Yaskawa INFORM job: DEMO_ROOF_SIDE_0625_3PAINT_32.JBI

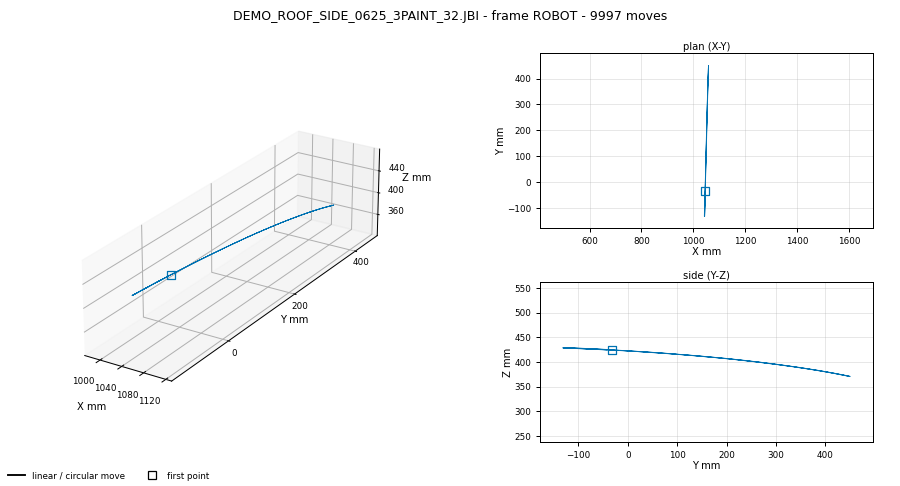
[picture p0: tool path of DEMO_ROOF_SIDE_0625_3PAINT_32.JBI in frame ROBOT, 9997 of 9997 moves have a stored position in this frame; points joined in program order, loops and branches not executed]
/JOB
//NAME DEMO_ROOF_SIDE_0625_3PAINT32
//POS
///NPOS 9997,0,0,0,0,0
///TOOL 0
///USER 0
///POSTYPE ROBOT
///RECTAN
///RCONF 1,0,0,0,0,0,0,0,0,0,0,0,0,0,0,0,0,0,0,0,0,0,0,0
C00000=1046.643,-32.584,425.197,169.918,33.552,156.330
C00001=1046.637,-32.833,425.210,169.916,33.551,156.330
C00002=1046.631,-33.082,425.224,169.914,33.549,156.330
C00003=1046.625,-33.331,425.237,169.912,33.548,156.330
C00004=1046.618,-33.581,425.250,169.910,33.547,156.329
C00005=1046.612,-33.831,425.264,169.908,33.546,156.329
C00006=1046.606,-34.081,425.276,169.906,33.544,156.329
C00007=1046.600,-34.330,425.290,169.904,33.543,156.329
C00008=1046.593,-34.580,425.303,169.902,33.542,156.329
C00009=1046.586,-34.860,425.319,169.899,33.541,156.329
C00010=1046.579,-35.141,425.334,169.897,33.539,156.329
C00011=1046.572,-35.422,425.348,169.895,33.538,156.328
C00012=1046.566,-35.702,425.363,169.893,33.536,156.328
C00013=1046.559,-35.952,425.377,169.891,33.535,156.328
C00014=1046.553,-36.202,425.389,169.889,33.534,156.328
C00015=1046.547,-36.451,425.403,169.887,33.533,156.328
C00016=1046.541,-36.700,425.416,169.885,33.531,156.328
C00017=1046.534,-36.950,425.429,169.883,33.530,156.327
C00018=1046.528,-37.200,425.442,169.881,33.529,156.327
C00019=1046.522,-37.450,425.455,169.879,33.528,156.327
C00020=1046.515,-37.699,425.469,169.877,33.526,156.327
C00021=1046.510,-37.949,425.481,169.875,33.525,156.327
C00022=1046.503,-38.198,425.494,169.873,33.524,156.327
C00023=1046.497,-38.447,425.508,169.870,33.523,156.326
C00024=1046.491,-38.698,425.521,169.868,33.521,156.326
C00025=1046.484,-38.947,425.534,169.866,33.520,156.326
C00026=1046.478,-39.196,425.547,169.864,33.519,156.326
C00027=1046.472,-39.446,425.560,169.862,33.518,156.326
C00028=1046.466,-39.695,425.573,169.860,33.517,156.326
C00029=1046.458,-39.945,425.586,169.858,33.515,156.326
C00030=1046.453,-40.195,425.599,169.856,33.515,156.325
C00031=1046.446,-40.444,425.612,169.854,33.513,156.325
C00032=1046.440,-40.694,425.624,169.852,33.512,156.325
C00033=1046.434,-40.943,425.638,169.850,33.511,156.325
C00034=1046.428,-41.193,425.650,169.848,33.510,156.325
C00035=1046.421,-41.443,425.663,169.846,33.509,156.325
C00036=1046.415,-41.692,425.677,169.844,33.507,156.325
C00037=1046.409,-41.942,425.689,169.842,33.507,156.324
C00038=1046.402,-42.191,425.702,169.840,33.505,156.324
C00039=1046.397,-42.441,425.715,169.838,33.504,156.324
C00040=1046.390,-42.690,425.728,169.836,33.503,156.324
C00041=1046.384,-42.940,425.740,169.834,33.502,156.324
C00042=1046.377,-43.189,425.753,169.832,33.501,156.324
C00043=1046.371,-43.440,425.766,169.830,33.500,156.324
C00044=1046.365,-43.689,425.780,169.827,33.498,156.324
C00045=1046.358,-43.939,425.792,169.825,33.497,156.323
C00046=1046.352,-44.188,425.805,169.823,33.496,156.323
C00047=1046.346,-44.438,425.817,169.821,33.495,156.323
C00048=1046.340,-44.687,425.831,169.819,33.494,156.323
C00049=1046.334,-44.937,425.843,169.817,33.493,156.323
C00050=1046.327,-45.187,425.855,169.815,33.492,156.323
C00051=1046.321,-45.436,425.868,169.813,33.490,156.323
C00052=1046.315,-45.686,425.881,169.811,33.490,156.322
C00053=1046.309,-45.935,425.894,169.809,33.488,156.322
C00054=1046.302,-46.185,425.906,169.807,33.487,156.322
C00055=1046.296,-46.435,425.919,169.805,33.486,156.322
C00056=1046.290,-46.684,425.932,169.803,33.485,156.322
C00057=1046.284,-46.934,425.945,169.801,33.484,156.322
C00058=1046.277,-47.183,425.958,169.799,33.483,156.322
C00059=1046.271,-47.433,425.970,169.797,33.482,156.321
C00060=1046.265,-47.683,425.983,169.794,33.481,156.321
C00061=1046.259,-47.932,425.996,169.792,33.479,156.321
C00062=1046.252,-48.182,426.008,169.790,33.478,156.321
C00063=1046.246,-48.432,426.021,169.788,33.477,156.321
C00064=1046.240,-48.681,426.034,169.786,33.476,156.321
C00065=1046.234,-48.931,426.046,169.784,33.475,156.321
C00066=1046.227,-49.181,426.058,169.782,33.474,156.321
C00067=1046.221,-49.430,426.072,169.780,33.473,156.320
C00068=1046.215,-49.680,426.084,169.778,33.472,156.320
C00069=1046.209,-49.930,426.097,169.776,33.470,156.320
C00070=1046.203,-50.179,426.109,169.774,33.470,156.320
C00071=1046.196,-50.428,426.122,169.772,33.469,156.320
C00072=1046.190,-50.678,426.134,169.769,33.467,156.320
C00073=1046.183,-50.959,426.148,169.767,33.466,156.320
C00074=1046.176,-51.241,426.162,169.765,33.465,156.320
C00075=1046.169,-51.521,426.176,169.763,33.464,156.320
C00076=1046.162,-51.803,426.190,169.761,33.463,156.319
C00077=1046.155,-52.052,426.202,169.759,33.462,156.319
C00078=1046.148,-52.302,426.214,169.757,33.461,156.319
C00079=1046.143,-52.552,426.227,169.755,33.460,156.319
C00080=1046.136,-52.801,426.239,169.752,33.459,156.319
C00081=1046.130,-53.051,426.252,169.750,33.458,156.319
C00082=1046.123,-53.300,426.264,169.748,33.457,156.319
C00083=1046.116,-53.550,426.276,169.746,33.456,156.319
C00084=1046.111,-53.800,426.288,169.744,33.456,156.319
C00085=1046.104,-54.049,426.300,169.742,33.455,156.319
C00086=1046.098,-54.299,426.313,169.740,33.453,156.318
C00087=1046.091,-54.549,426.325,169.738,33.453,156.318
C00088=1046.085,-54.798,426.337,169.735,33.452,156.318
C00089=1046.079,-55.048,426.349,169.733,33.451,156.318
C00090=1046.073,-55.297,426.361,169.731,33.450,156.318
C00091=1046.067,-55.547,426.373,169.729,33.449,156.318
C00092=1046.060,-55.796,426.386,169.727,33.448,156.318
C00093=1046.053,-56.045,426.398,169.725,33.447,156.318
C00094=1046.047,-56.295,426.411,169.723,33.446,156.318
C00095=1046.041,-56.545,426.423,169.720,33.445,156.318
C00096=1046.034,-56.795,426.435,169.718,33.444,156.317
C00097=1046.028,-57.044,426.447,169.716,33.443,156.317
C00098=1046.021,-57.294,426.459,169.714,33.442,156.317
C00099=1046.016,-57.544,426.472,169.712,33.442,156.317
C00100=1046.009,-57.793,426.484,169.710,33.441,156.317
C00101=1046.002,-58.043,426.496,169.708,33.439,156.317
C00102=1045.997,-58.293,426.507,169.705,33.439,156.317
C00103=1045.991,-58.542,426.519,169.703,33.438,156.317
C00104=1045.984,-58.792,426.531,169.701,33.437,156.317
C00105=1045.978,-59.042,426.543,169.699,33.436,156.317
C00106=1045.971,-59.291,426.555,169.697,33.435,156.317
C00107=1045.965,-59.541,426.567,169.695,33.434,156.316
C00108=1045.959,-59.791,426.580,169.693,33.433,156.316
C00109=1045.953,-60.040,426.592,169.690,33.432,156.316
C00110=1045.947,-60.290,426.604,169.688,33.431,156.316
C00111=1045.940,-60.539,426.616,169.686,33.431,156.316
C00112=1045.934,-60.789,426.628,169.684,33.430,156.316
C00113=1045.928,-61.039,426.641,169.682,33.428,156.316
C00114=1045.921,-61.289,426.652,169.680,33.428,156.316
C00115=1045.915,-61.538,426.663,169.677,33.427,156.316
C00116=1045.909,-61.788,426.676,169.675,33.426,156.316
C00117=1045.903,-62.037,426.688,169.673,33.425,156.316
C00118=1045.896,-62.287,426.700,169.671,33.424,156.316
C00119=1045.889,-62.536,426.712,169.669,33.424,156.315
C00120=1045.884,-62.786,426.723,169.667,33.423,156.315
C00121=1045.878,-63.036,426.735,169.665,33.421,156.315
C00122=1045.871,-63.285,426.747,169.662,33.420,156.315
C00123=1045.865,-63.535,426.760,169.660,33.420,156.315
C00124=1045.859,-63.784,426.771,169.658,33.419,156.315
C00125=1045.853,-64.034,426.783,169.656,33.418,156.315
C00126=1045.847,-64.284,426.795,169.654,33.417,156.315
C00127=1045.840,-64.534,426.807,169.652,33.416,156.315
C00128=1045.834,-64.783,426.819,169.649,33.416,156.315
C00129=1045.829,-65.033,426.831,169.647,33.415,156.315
C00130=1045.822,-65.283,426.843,169.645,33.413,156.314
C00131=1045.815,-65.532,426.854,169.643,33.413,156.314
C00132=1045.809,-65.781,426.866,169.642,33.412,156.314
C00133=1045.804,-66.032,426.878,169.640,33.411,156.314
C00134=1045.797,-66.281,426.890,169.637,33.410,156.314
C00135=1045.791,-66.530,426.901,169.635,33.409,156.314
C00136=1045.785,-66.780,426.913,169.633,33.409,156.314
C00137=1045.778,-67.063,426.927,169.631,33.408,156.314
C00138=1045.772,-67.345,426.940,169.628,33.407,156.314
C00139=1045.765,-67.627,426.954,169.626,33.405,156.314
C00140=1045.757,-67.910,426.966,169.623,33.405,156.314
C00141=1045.751,-68.160,426.979,169.621,33.404,156.314
C00142=1045.745,-68.410,426.990,169.619,33.403,156.314
C00143=1045.739,-68.659,427.002,169.617,33.402,156.313
C00144=1045.733,-68.908,427.014,169.614,33.401,156.313
C00145=1045.727,-69.159,427.025,169.612,33.400,156.313
C00146=1045.721,-69.408,427.037,169.610,33.400,156.313
C00147=1045.714,-69.658,427.048,169.608,33.399,156.313
C00148=1045.708,-69.908,427.061,169.606,33.398,156.313
C00149=1045.702,-70.156,427.072,169.604,33.397,156.313
C00150=1045.696,-70.407,427.084,169.601,33.396,156.313
C00151=1045.690,-70.656,427.095,169.599,33.396,156.313
C00152=1045.684,-70.906,427.107,169.597,33.395,156.313
C00153=1045.678,-71.156,427.119,169.595,33.394,156.313
C00154=1045.672,-71.405,427.130,169.593,33.393,156.313
C00155=1045.665,-71.655,427.142,169.590,33.392,156.313
C00156=1045.660,-71.904,427.153,169.588,33.391,156.313
C00157=1045.654,-72.154,427.165,169.586,33.391,156.312
C00158=1045.647,-72.404,427.176,169.584,33.390,156.312
C00159=1045.641,-72.653,427.188,169.582,33.389,156.312
C00160=1045.635,-72.903,427.199,169.579,33.388,156.312
C00161=1045.630,-73.152,427.211,169.577,33.387,156.312
C00162=1045.623,-73.403,427.223,169.575,33.387,156.312
C00163=1045.617,-73.652,427.234,169.573,33.386,156.312
C00164=1045.611,-73.902,427.246,169.571,33.385,156.312
C00165=1045.605,-74.151,427.257,169.568,33.384,156.312
C00166=1045.598,-74.401,427.268,169.566,33.383,156.312
C00167=1045.592,-74.651,427.280,169.564,33.382,156.312
C00168=1045.586,-74.900,427.291,169.562,33.382,156.312
C00169=1045.580,-75.150,427.302,169.560,33.382,156.312
C00170=1045.574,-75.400,427.313,169.557,33.381,156.312
C00171=1045.567,-75.649,427.325,169.555,33.380,156.312
C00172=1045.561,-75.899,427.337,169.553,33.379,156.312
C00173=1045.555,-76.148,427.348,169.551,33.378,156.311
C00174=1045.549,-76.398,427.359,169.548,33.378,156.311
C00175=1045.543,-76.648,427.370,169.546,33.377,156.311
C00176=1045.537,-76.898,427.381,169.544,33.376,156.311
C00177=1045.530,-77.147,427.393,169.542,33.376,156.311
C00178=1045.524,-77.397,427.404,169.540,33.375,156.311
C00179=1045.518,-77.647,427.415,169.538,33.375,156.311
C00180=1045.512,-77.896,427.427,169.536,33.374,156.311
C00181=1045.506,-78.146,427.438,169.534,33.373,156.311
C00182=1045.500,-78.396,427.449,169.532,33.372,156.311
C00183=1045.494,-78.645,427.460,169.529,33.372,156.311
C00184=1045.487,-78.895,427.472,169.527,33.371,156.311
C00185=1045.482,-79.144,427.483,169.525,33.370,156.311
C00186=1045.475,-79.395,427.494,169.523,33.369,156.311
C00187=1045.469,-79.644,427.505,169.520,33.369,156.311
C00188=1045.462,-79.893,427.516,169.518,33.368,156.311
C00189=1045.456,-80.143,427.527,169.516,33.368,156.311
C00190=1045.450,-80.393,427.539,169.514,33.367,156.311
C00191=1045.444,-80.643,427.550,169.511,33.367,156.311
C00192=1045.437,-80.892,427.560,169.509,33.366,156.311
C00193=1045.431,-81.143,427.571,169.507,33.366,156.311
C00194=1045.425,-81.392,427.582,169.505,33.365,156.311
C00195=1045.418,-81.642,427.594,169.502,33.364,156.311
C00196=1045.412,-81.891,427.605,169.500,33.364,156.311
C00197=1045.406,-82.141,427.616,169.498,33.364,156.311
C00198=1045.400,-82.390,427.627,169.495,33.363,156.311
C00199=1045.393,-82.640,427.637,169.493,33.362,156.311
C00200=1045.387,-82.890,427.648,169.491,33.362,156.311
C00201=1045.380,-83.174,427.661,169.488,33.361,156.311
C00202=1045.373,-83.459,427.673,169.486,33.361,156.311
C00203=1045.366,-83.743,427.686,169.483,33.360,156.311
C00204=1045.358,-84.029,427.698,169.481,33.360,156.311
C00205=1045.353,-84.278,427.709,169.478,33.359,156.311
C00206=1045.346,-84.528,427.720,169.476,33.358,156.311
C00207=1045.340,-84.777,427.730,169.474,33.358,156.310
C00208=1045.334,-85.027,427.741,169.471,33.357,156.311
C00209=1045.328,-85.277,427.753,169.469,33.357,156.310
C00210=1045.321,-85.526,427.763,169.467,33.356,156.310
C00211=1045.315,-85.777,427.774,169.465,33.356,156.310
C00212=1045.309,-86.026,427.785,169.462,33.355,156.310
C00213=1045.303,-86.275,427.795,169.460,33.355,156.310
C00214=1045.296,-86.525,427.807,169.459,33.354,156.310
C00215=1045.291,-86.775,427.817,169.456,33.354,156.310
C00216=1045.284,-87.025,427.828,169.454,33.353,156.310
C00217=1045.278,-87.274,427.839,169.452,33.353,156.310
C00218=1045.272,-87.524,427.850,169.450,33.352,156.310
C00219=1045.265,-87.774,427.860,169.447,33.352,156.310
C00220=1045.259,-88.023,427.871,169.445,33.351,156.310
C00221=1045.253,-88.273,427.882,169.443,33.351,156.310
C00222=1045.246,-88.522,427.893,169.440,33.350,156.310
C00223=1045.241,-88.773,427.903,169.438,33.349,156.310
C00224=1045.234,-89.022,427.914,169.436,33.349,156.310
C00225=1045.228,-89.272,427.925,169.434,33.348,156.310
C00226=1045.222,-89.521,427.935,169.431,33.348,156.310
C00227=1045.216,-89.771,427.946,169.429,33.348,156.310
C00228=1045.210,-90.021,427.957,169.427,33.347,156.310
C00229=1045.204,-90.270,427.968,169.424,33.347,156.310
C00230=1045.198,-90.520,427.977,169.422,33.346,156.310
C00231=1045.191,-90.770,427.989,169.420,33.346,156.310
C00232=1045.186,-91.020,427.999,169.418,33.345,156.310
C00233=1045.179,-91.269,428.010,169.415,33.345,156.310
C00234=1045.173,-91.519,428.021,169.413,33.345,156.310
C00235=1045.166,-91.768,428.031,169.411,33.344,156.310
C00236=1045.161,-92.018,428.041,169.408,33.344,156.310
C00237=1045.155,-92.268,428.052,169.406,33.343,156.310
C00238=1045.148,-92.518,428.063,169.404,33.343,156.310
C00239=1045.142,-92.767,428.074,169.401,33.343,156.310
C00240=1045.136,-93.017,428.083,169.399,33.342,156.310
C00241=1045.130,-93.267,428.094,169.397,33.342,156.310
C00242=1045.124,-93.517,428.106,169.395,33.341,156.310
C00243=1045.118,-93.766,428.116,169.392,33.340,156.310
C00244=1045.112,-94.016,428.126,169.390,33.340,156.310
C00245=1045.106,-94.266,428.137,169.388,33.340,156.310
C00246=1045.099,-94.515,428.148,169.385,33.339,156.310
C00247=1045.094,-94.766,428.158,169.383,33.339,156.310
C00248=1045.087,-95.015,428.168,169.382,33.338,156.310
C00249=1045.082,-95.264,428.179,169.379,33.338,156.310
C00250=1045.076,-95.514,428.188,169.377,33.337,156.310
C00251=1045.069,-95.764,428.200,169.375,33.337,156.310
C00252=1045.063,-96.014,428.211,169.373,33.337,156.310
C00253=1045.057,-96.263,428.220,169.370,33.336,156.310
C00254=1045.052,-96.513,428.231,169.368,33.336,156.310
C00255=1045.045,-96.762,428.241,169.366,33.336,156.310
C00256=1045.040,-97.012,428.251,169.363,33.335,156.310
C00257=1045.033,-97.262,428.262,169.361,33.335,156.310
C00258=1045.027,-97.512,428.272,169.359,33.334,156.310
C00259=1045.021,-97.761,428.283,169.356,33.334,156.310
C00260=1045.015,-98.011,428.293,169.354,33.334,156.310
C00261=1045.009,-98.261,428.303,169.352,33.333,156.310
C00262=1045.002,-98.511,428.314,169.349,33.333,156.310
C00263=1044.996,-98.761,428.324,169.347,33.333,156.311
C00264=1044.990,-99.010,428.334,169.345,33.333,156.311
C00265=1044.982,-99.297,428.345,169.342,33.332,156.311
C00266=1044.976,-99.583,428.357,169.339,33.332,156.311
C00267=1044.969,-99.871,428.369,169.337,33.331,156.311
C00268=1044.961,-100.158,428.381,169.334,33.331,156.311
C00269=1044.956,-100.408,428.391,169.332,33.331,156.311
C00270=1044.949,-100.657,428.401,169.329,33.331,156.311
C00271=1044.943,-100.907,428.411,169.327,33.330,156.311
C00272=1044.937,-101.157,428.422,169.325,33.330,156.311
C00273=1044.931,-101.407,428.431,169.322,33.330,156.311
C00274=1044.924,-101.656,428.442,169.320,33.330,156.311
C00275=1044.919,-101.906,428.452,169.318,33.330,156.311
C00276=1044.913,-102.156,428.461,169.315,33.329,156.311
C00277=1044.906,-102.405,428.472,169.313,33.329,156.311
C00278=1044.901,-102.655,428.482,169.310,33.328,156.311
C00279=1044.894,-102.904,428.492,169.309,33.328,156.311
C00280=1044.888,-103.154,428.502,169.307,33.328,156.311
C00281=1044.882,-103.404,428.511,169.304,33.328,156.311
C00282=1044.875,-103.654,428.523,169.302,33.328,156.311
C00283=1044.869,-103.904,428.532,169.300,33.327,156.311
C00284=1044.863,-104.154,428.542,169.297,33.327,156.311
C00285=1044.857,-104.403,428.553,169.295,33.327,156.311
C00286=1044.851,-104.653,428.562,169.293,33.327,156.311
C00287=1044.845,-104.903,428.572,169.290,33.327,156.311
C00288=1044.839,-105.152,428.582,169.288,33.326,156.311
C00289=1044.833,-105.402,428.592,169.286,33.326,156.311
C00290=1044.827,-105.652,428.602,169.283,33.326,156.312
C00291=1044.820,-105.901,428.612,169.281,33.326,156.312
C00292=1044.814,-106.151,428.622,169.279,33.326,156.312
C00293=1044.809,-106.401,428.632,169.276,33.325,156.312
C00294=1044.803,-106.651,428.641,169.274,33.325,156.312
C00295=1044.796,-106.900,428.652,169.272,33.325,156.312
C00296=1044.790,-107.150,428.661,169.269,33.325,156.312
C00297=1044.785,-107.400,428.671,169.267,33.325,156.312
C00298=1044.778,-107.649,428.681,169.264,33.324,156.312
C00299=1044.772,-107.899,428.691,169.262,33.324,156.312
C00300=1044.766,-108.148,428.701,169.260,33.324,156.312
C00301=1044.760,-108.398,428.710,169.257,33.324,156.312
C00302=1044.753,-108.648,428.720,169.255,33.324,156.312
C00303=1044.747,-108.898,428.729,169.253,33.324,156.312
C00304=1044.741,-109.147,428.740,169.250,33.324,156.312
C00305=1044.735,-109.397,428.749,169.248,33.324,156.312
C00306=1044.728,-109.647,428.759,169.245,33.323,156.312
C00307=1044.723,-109.897,428.769,169.243,33.323,156.312
C00308=1044.717,-110.146,428.779,169.242,33.324,156.313
C00309=1044.711,-110.396,428.788,169.239,33.323,156.313
C00310=1044.705,-110.646,428.798,169.237,33.323,156.313
C00311=1044.698,-110.896,428.807,169.235,33.323,156.313
C00312=1044.692,-111.145,428.818,169.232,33.323,156.313
C00313=1044.686,-111.395,428.827,169.230,33.323,156.313
C00314=1044.680,-111.645,428.837,169.227,33.323,156.313
C00315=1044.673,-111.894,428.846,169.225,33.323,156.313
C00316=1044.667,-112.144,428.856,169.223,33.323,156.313
C00317=1044.661,-112.394,428.865,169.220,33.322,156.313
C00318=1044.655,-112.644,428.875,169.218,33.322,156.313
C00319=1044.649,-112.894,428.885,169.216,33.323,156.313
C00320=1044.643,-113.144,428.895,169.213,33.322,156.313
C00321=1044.637,-113.394,428.904,169.211,33.322,156.313
C00322=1044.631,-113.643,428.914,169.208,33.322,156.313
C00323=1044.625,-113.892,428.923,169.206,33.322,156.313
C00324=1044.619,-114.142,428.933,169.204,33.322,156.314
C00325=1044.613,-114.392,428.942,169.201,33.322,156.314
C00326=1044.607,-114.642,428.952,169.199,33.322,156.314
C00327=1044.601,-114.892,428.961,169.196,33.322,156.314
C00328=1044.594,-115.141,428.971,169.194,33.322,156.314
C00329=1044.587,-115.427,428.982,169.191,33.322,156.314
C00330=1044.581,-115.713,428.992,169.189,33.322,156.314
C00331=1044.573,-115.999,429.003,169.186,33.322,156.314
C00332=1044.566,-116.285,429.014,169.183,33.322,156.314
C00333=1044.561,-116.534,429.023,169.181,33.322,156.314
C00334=1044.554,-116.784,429.033,169.178,33.322,156.314
C00335=1044.548,-117.034,429.043,169.177,33.322,156.315
C00336=1044.542,-117.284,429.052,169.175,33.322,156.315
C00337=1044.536,-117.534,429.061,169.172,33.322,156.315
C00338=1044.529,-117.784,429.070,169.170,33.323,156.315
C00339=1044.523,-118.033,429.080,169.167,33.322,156.315
C00340=1044.518,-118.283,429.089,169.165,33.322,156.315
C00341=1044.511,-118.532,429.098,169.163,33.323,156.315
C00342=1044.505,-118.782,429.108,169.160,33.322,156.315
C00343=1044.499,-119.033,429.117,169.158,33.323,156.315
C00344=1044.493,-119.282,429.126,169.155,33.323,156.315
C00345=1044.487,-119.532,429.136,169.153,33.322,156.315
C00346=1044.481,-119.781,429.144,169.150,33.323,156.316
C00347=1044.474,-120.031,429.154,169.148,33.323,156.316
C00348=1044.469,-120.281,429.163,169.146,33.323,156.316
C00349=1044.462,-120.531,429.172,169.143,33.323,156.316
C00350=1044.456,-120.781,429.182,169.141,33.323,156.316
C00351=1044.451,-121.030,429.191,169.138,33.323,156.316
C00352=1044.445,-121.280,429.200,169.136,33.323,156.316
C00353=1044.438,-121.530,429.209,169.134,33.323,156.316
C00354=1044.432,-121.780,429.219,169.131,33.324,156.316
C00355=1044.426,-122.029,429.228,169.129,33.323,156.316
C00356=1044.420,-122.279,429.237,169.126,33.324,156.317
C00357=1044.414,-122.529,429.246,169.124,33.324,156.317
C00358=1044.408,-122.779,429.256,169.122,33.324,156.317
C00359=1044.402,-123.028,429.264,169.119,33.324,156.317
C00360=1044.396,-123.278,429.273,169.117,33.324,156.317
C00361=1044.390,-123.528,429.283,169.114,33.324,156.317
C00362=1044.384,-123.778,429.292,169.113,33.325,156.317
C00363=1044.378,-124.027,429.301,169.111,33.324,156.317
C00364=1044.371,-124.277,429.310,169.108,33.325,156.317
C00365=1044.365,-124.527,429.319,169.106,33.325,156.317
C00366=1044.359,-124.777,429.328,169.103,33.325,156.318
C00367=1044.354,-125.026,429.337,169.101,33.325,156.318
C00368=1044.347,-125.276,429.346,169.098,33.325,156.318
C00369=1044.341,-125.526,429.355,169.096,33.326,156.318
C00370=1044.335,-125.776,429.364,169.094,33.326,156.318
C00371=1044.329,-126.025,429.373,169.091,33.326,156.318
C00372=1044.323,-126.275,429.382,169.089,33.326,156.318
C00373=1044.317,-126.525,429.391,169.086,33.326,156.318
C00374=1044.310,-126.774,429.400,169.084,33.327,156.319
C00375=1044.305,-127.025,429.409,169.081,33.327,156.319
C00376=1044.298,-127.274,429.418,169.079,33.327,156.319
C00377=1044.292,-127.524,429.426,169.077,33.327,156.319
C00378=1044.286,-127.774,429.436,169.074,33.328,156.319
C00379=1044.281,-128.023,429.445,169.072,33.328,156.319
C00380=1044.277,-128.273,429.455,169.070,33.327,156.319
C00381=1044.273,-128.523,429.465,169.067,33.326,156.319
C00382=1044.270,-128.773,429.476,169.065,33.324,156.319
C00383=1044.268,-129.022,429.488,169.064,33.322,156.318
C00384=1044.267,-129.272,429.501,169.062,33.320,156.318
C00385=1044.267,-129.523,429.514,169.060,33.317,156.318
C00386=1044.268,-129.773,429.528,169.059,33.314,156.317
C00387=1044.270,-130.023,429.541,169.057,33.310,156.317
C00388=1044.272,-130.274,429.556,169.056,33.306,156.316
C00389=1044.276,-130.524,429.572,169.055,33.301,156.315
C00390=1044.281,-130.774,429.588,169.054,33.296,156.314
C00391=1044.286,-131.025,429.605,169.053,33.290,156.313
C00392=1044.292,-131.275,429.623,169.052,33.284,156.312
C00393=1043.938,-131.299,429.377,169.006,33.467,156.345
C00394=1043.932,-131.048,429.360,169.007,33.473,156.346
C00395=1043.927,-130.798,429.343,169.008,33.479,156.347
C00396=1043.922,-130.548,429.327,169.009,33.484,156.348
C00397=1043.918,-130.297,429.312,169.010,33.489,156.349
C00398=1043.916,-130.047,429.296,169.011,33.493,156.349
C00399=1043.914,-129.797,429.282,169.012,33.497,156.350
C00400=1043.914,-129.547,429.268,169.014,33.500,156.350
C00401=1043.914,-129.296,429.255,169.015,33.503,156.351
C00402=1043.914,-129.046,429.243,169.017,33.506,156.351
C00403=1043.915,-128.796,429.231,169.019,33.508,156.352
C00404=1043.919,-128.546,429.220,169.021,33.509,156.352
C00405=1043.922,-128.296,429.209,169.023,33.510,156.352
C00406=1043.927,-128.047,429.199,169.025,33.511,156.352
C00407=1043.932,-127.797,429.189,169.028,33.511,156.352
C00408=1043.938,-127.547,429.181,169.030,33.510,156.352
C00409=1043.944,-127.298,429.172,169.032,33.510,156.351
C00410=1043.950,-127.048,429.162,169.035,33.510,156.351
C00411=1043.956,-126.799,429.154,169.037,33.510,156.351
C00412=1043.962,-126.549,429.145,169.040,33.509,156.351
C00413=1043.968,-126.299,429.136,169.042,33.509,156.351
C00414=1043.975,-126.049,429.127,169.045,33.509,156.351
C00415=1043.980,-125.799,429.119,169.047,33.509,156.351
C00416=1043.986,-125.550,429.109,169.050,33.509,156.351
C00417=1043.993,-125.300,429.100,169.052,33.508,156.351
C00418=1043.999,-125.050,429.092,169.054,33.508,156.350
C00419=1044.005,-124.801,429.082,169.057,33.508,156.350
C00420=1044.011,-124.551,429.074,169.059,33.508,156.350
C00421=1044.018,-124.301,429.064,169.062,33.507,156.350
C00422=1044.023,-124.052,429.055,169.064,33.507,156.350
C00423=1044.029,-123.801,429.046,169.067,33.507,156.350
C00424=1044.035,-123.551,429.037,169.069,33.507,156.350
C00425=1044.042,-123.302,429.028,169.071,33.507,156.350
C00426=1044.047,-123.052,429.019,169.074,33.507,156.350
C00427=1044.054,-122.802,429.010,169.076,33.506,156.349
C00428=1044.060,-122.553,429.000,169.079,33.507,156.349
C00429=1044.066,-122.302,428.991,169.080,33.506,156.349
C00430=1044.072,-122.053,428.983,169.083,33.506,156.349
C00431=1044.078,-121.804,428.973,169.085,33.506,156.349
C00432=1044.084,-121.553,428.964,169.087,33.506,156.349
C00433=1044.090,-121.303,428.955,169.090,33.506,156.349
C00434=1044.096,-121.054,428.945,169.092,33.505,156.349
C00435=1044.102,-120.805,428.936,169.095,33.505,156.349
C00436=1044.108,-120.554,428.927,169.097,33.506,156.349
C00437=1044.115,-120.305,428.918,169.100,33.505,156.348
C00438=1044.121,-120.055,428.908,169.102,33.505,156.348
C00439=1044.126,-119.806,428.899,169.104,33.505,156.348
C00440=1044.132,-119.556,428.890,169.107,33.505,156.348
C00441=1044.138,-119.306,428.881,169.109,33.505,156.348
C00442=1044.145,-119.056,428.871,169.112,33.505,156.348
C00443=1044.151,-118.806,428.862,169.114,33.504,156.348
C00444=1044.157,-118.557,428.853,169.116,33.505,156.348
C00445=1044.163,-118.307,428.843,169.119,33.504,156.348
C00446=1044.169,-118.057,428.835,169.121,33.504,156.348
C00447=1044.175,-117.807,428.825,169.124,33.505,156.348
C00448=1044.181,-117.557,428.815,169.126,33.504,156.347
C00449=1044.188,-117.308,428.806,169.128,33.504,156.347
C00450=1044.193,-117.058,428.797,169.131,33.504,156.347
C00451=1044.199,-116.809,428.787,169.133,33.504,156.347
C00452=1044.205,-116.559,428.778,169.136,33.504,156.347
C00453=1044.212,-116.309,428.768,169.138,33.504,156.347
C00454=1044.219,-116.023,428.758,169.141,33.504,156.347
C00455=1044.226,-115.738,428.747,169.143,33.504,156.347
C00456=1044.233,-115.451,428.736,169.145,33.504,156.347
C00457=1044.240,-115.165,428.725,169.148,33.504,156.347
C00458=1044.246,-114.915,428.716,169.151,33.504,156.347
C00459=1044.252,-114.665,428.706,169.153,33.504,156.346
C00460=1044.258,-114.416,428.697,169.155,33.504,156.346
C00461=1044.264,-114.166,428.687,169.158,33.504,156.346
C00462=1044.270,-113.916,428.678,169.160,33.504,156.346
C00463=1044.276,-113.667,428.668,169.163,33.504,156.346
C00464=1044.282,-113.417,428.659,169.165,33.503,156.346
C00465=1044.288,-113.167,428.649,169.167,33.504,156.346
C00466=1044.295,-112.917,428.640,169.170,33.504,156.346
C00467=1044.301,-112.667,428.630,169.172,33.504,156.346
C00468=1044.307,-112.418,428.620,169.175,33.504,156.346
C00469=1044.313,-112.168,428.610,169.177,33.504,156.346
C00470=1044.320,-111.919,428.601,169.179,33.504,156.346
C00471=1044.326,-111.669,428.591,169.182,33.504,156.346
C00472=1044.331,-111.420,428.582,169.184,33.504,156.346
C00473=1044.337,-111.170,428.572,169.186,33.504,156.345
C00474=1044.343,-110.920,428.562,169.189,33.504,156.345
C00475=1044.349,-110.670,428.553,169.191,33.504,156.345
C00476=1044.355,-110.420,428.543,169.194,33.504,156.345
C00477=1044.361,-110.170,428.533,169.196,33.505,156.345
C00478=1044.368,-109.921,428.524,169.198,33.504,156.345
C00479=1044.374,-109.671,428.514,169.201,33.504,156.345
C00480=1044.380,-109.422,428.504,169.203,33.505,156.345
C00481=1044.386,-109.172,428.494,169.206,33.505,156.345
C00482=1044.393,-108.922,428.485,169.208,33.505,156.345
C00483=1044.399,-108.672,428.475,169.210,33.504,156.345
C00484=1044.404,-108.422,428.465,169.212,33.505,156.345
C00485=1044.410,-108.172,428.456,169.214,33.505,156.345
C00486=1044.417,-107.923,428.445,169.216,33.505,156.345
C00487=1044.423,-107.673,428.436,169.219,33.505,156.345
C00488=1044.429,-107.424,428.426,169.221,33.505,156.345
C00489=1044.435,-107.174,428.417,169.224,33.506,156.345
C00490=1044.442,-106.925,428.406,169.226,33.506,156.344
C00491=1044.447,-106.674,428.396,169.228,33.505,156.344
C00492=1044.453,-106.425,428.387,169.231,33.506,156.344
C00493=1044.460,-106.175,428.377,169.233,33.506,156.344
C00494=1044.466,-105.926,428.367,169.235,33.506,156.344
C00495=1044.472,-105.675,428.356,169.238,33.506,156.344
C00496=1044.478,-105.425,428.347,169.240,33.506,156.344
C00497=1044.485,-105.175,428.337,169.243,33.507,156.344
C00498=1044.491,-104.926,428.327,169.245,33.507,156.344
C00499=1044.496,-104.676,428.317,169.247,33.507,156.344
C00500=1044.503,-104.426,428.307,169.250,33.507,156.344
C00501=1044.509,-104.177,428.297,169.252,33.507,156.344
C00502=1044.515,-103.927,428.287,169.254,33.507,156.344
C00503=1044.521,-103.677,428.277,169.257,33.508,156.344
C00504=1044.527,-103.428,428.267,169.259,33.508,156.344
C00505=1044.533,-103.178,428.257,169.261,33.508,156.344
C00506=1044.539,-102.929,428.246,169.264,33.508,156.344
C00507=1044.545,-102.679,428.237,169.266,33.508,156.344
C00508=1044.551,-102.429,428.227,169.269,33.509,156.344
C00509=1044.558,-102.179,428.216,169.271,33.509,156.344
C00510=1044.564,-101.929,428.206,169.273,33.509,156.343
C00511=1044.570,-101.680,428.196,169.276,33.510,156.344
C00512=1044.576,-101.430,428.186,169.278,33.510,156.344
C00513=1044.582,-101.180,428.176,169.280,33.510,156.343
C00514=1044.588,-100.931,428.166,169.283,33.510,156.343
C00515=1044.595,-100.681,428.157,169.284,33.511,156.343
C00516=1044.600,-100.431,428.146,169.286,33.511,156.343
C00517=1044.607,-100.181,428.136,169.289,33.511,156.343
C00518=1044.614,-99.895,428.124,169.291,33.511,156.343
C00519=1044.621,-99.607,428.112,169.294,33.511,156.343
C00520=1044.628,-99.321,428.100,169.297,33.512,156.343
C00521=1044.636,-99.033,428.089,169.300,33.512,156.343
C00522=1044.641,-98.784,428.078,169.302,33.512,156.343
C00523=1044.648,-98.534,428.069,169.304,33.513,156.343
C00524=1044.654,-98.285,428.058,169.307,33.513,156.343
C00525=1044.660,-98.035,428.048,169.309,33.513,156.343
C00526=1044.667,-97.785,428.038,169.311,33.513,156.343
C00527=1044.673,-97.536,428.027,169.314,33.514,156.343
C00528=1044.678,-97.286,428.017,169.316,33.514,156.343
C00529=1044.684,-97.036,428.006,169.318,33.515,156.343
C00530=1044.690,-96.786,427.997,169.321,33.515,156.343
C00531=1044.696,-96.537,427.986,169.323,33.515,156.343
C00532=1044.703,-96.287,427.975,169.325,33.515,156.343
C00533=1044.709,-96.037,427.965,169.328,33.516,156.343
C00534=1044.715,-95.788,427.955,169.330,33.516,156.343
C00535=1044.721,-95.538,427.944,169.332,33.516,156.343
C00536=1044.726,-95.288,427.934,169.334,33.517,156.343
C00537=1044.733,-95.038,427.923,169.337,33.517,156.343
C00538=1044.739,-94.789,427.912,169.339,33.518,156.343
C00539=1044.745,-94.539,427.903,169.341,33.518,156.343
C00540=1044.751,-94.289,427.892,169.344,33.519,156.343
C00541=1044.757,-94.040,427.881,169.346,33.519,156.343
C00542=1044.764,-93.789,427.871,169.348,33.520,156.343
C00543=1044.769,-93.540,427.860,169.351,33.520,156.343
C00544=1044.776,-93.291,427.850,169.353,33.520,156.343
C00545=1044.782,-93.041,427.839,169.355,33.521,156.343
C00546=1044.788,-92.790,427.828,169.358,33.521,156.343
C00547=1044.794,-92.541,427.818,169.360,33.521,156.343
C00548=1044.800,-92.292,427.807,169.362,33.522,156.343
C00549=1044.806,-92.043,427.797,169.364,33.522,156.343
C00550=1044.812,-91.792,427.786,169.366,33.523,156.343
C00551=1044.818,-91.542,427.775,169.368,33.523,156.343
C00552=1044.824,-91.293,427.765,169.370,33.523,156.343
C00553=1044.831,-91.043,427.754,169.373,33.524,156.343
C00554=1044.837,-90.793,427.743,169.375,33.524,156.343
C00555=1044.843,-90.544,427.733,169.377,33.525,156.343
C00556=1044.848,-90.294,427.723,169.380,33.525,156.343
C00557=1044.856,-90.044,427.712,169.382,33.526,156.343
C00558=1044.861,-89.795,427.701,169.384,33.526,156.343
C00559=1044.867,-89.545,427.690,169.387,33.527,156.343
C00560=1044.874,-89.295,427.680,169.389,33.527,156.343
C00561=1044.880,-89.046,427.669,169.391,33.528,156.343
C00562=1044.885,-88.796,427.659,169.393,33.528,156.343
C00563=1044.892,-88.546,427.648,169.396,33.529,156.343
C00564=1044.898,-88.296,427.637,169.398,33.529,156.343
C00565=1044.904,-88.047,427.626,169.400,33.530,156.343
C00566=1044.911,-87.797,427.616,169.403,33.530,156.343
C00567=1044.917,-87.548,427.605,169.405,33.530,156.343
C00568=1044.922,-87.298,427.594,169.407,33.531,156.343
C00569=1044.929,-87.048,427.583,169.410,33.531,156.343
C00570=1044.935,-86.799,427.572,169.412,33.532,156.343
C00571=1044.942,-86.549,427.561,169.414,33.532,156.343
C00572=1044.948,-86.299,427.551,169.416,33.533,156.343
C00573=1044.954,-86.050,427.540,169.419,33.533,156.343
C00574=1044.960,-85.800,427.529,169.421,33.534,156.343
C00575=1044.967,-85.550,427.518,169.423,33.534,156.343
C00576=1044.973,-85.300,427.507,169.426,33.534,156.343
C00577=1044.979,-85.051,427.496,169.428,33.535,156.343
C00578=1044.985,-84.802,427.486,169.430,33.535,156.343
C00579=1044.991,-84.551,427.475,169.432,33.536,156.343
C00580=1044.997,-84.302,427.464,169.435,33.536,156.343
C00581=1045.004,-84.052,427.453,169.437,33.537,156.343
C00582=1045.011,-83.767,427.441,169.440,33.537,156.343
C00583=1045.019,-83.483,427.428,169.442,33.538,156.343
C00584=1045.025,-83.198,427.416,169.445,33.539,156.343
C00585=1045.033,-82.913,427.403,169.447,33.539,156.343
C00586=1045.039,-82.664,427.392,169.450,33.540,156.343
C00587=1045.045,-82.414,427.381,169.452,33.540,156.343
C00588=1045.052,-82.164,427.371,169.454,33.541,156.343
C00589=1045.057,-81.915,427.360,169.456,33.541,156.343
C00590=1045.064,-81.665,427.349,169.458,33.542,156.343
C00591=1045.069,-81.415,427.338,169.460,33.542,156.343
C00592=1045.076,-81.165,427.327,169.462,33.543,156.343
C00593=1045.083,-80.916,427.315,169.465,33.543,156.343
C00594=1045.089,-80.666,427.304,169.467,33.544,156.343
C00595=1045.095,-80.416,427.293,169.469,33.544,156.343
C00596=1045.102,-80.167,427.283,169.471,33.545,156.343
C00597=1045.108,-79.917,427.272,169.474,33.546,156.343
C00598=1045.114,-79.667,427.261,169.476,33.546,156.343
C00599=1045.120,-79.418,427.249,169.478,33.547,156.343
C00600=1045.126,-79.168,427.238,169.481,33.548,156.343
C00601=1045.132,-78.918,427.227,169.483,33.548,156.343
C00602=1045.138,-78.669,427.216,169.485,33.548,156.343
C00603=1045.145,-78.419,427.204,169.487,33.549,156.344
C00604=1045.151,-78.169,427.193,169.489,33.549,156.344
C00605=1045.158,-77.920,427.182,169.492,33.550,156.344
C00606=1045.163,-77.670,427.171,169.494,33.551,156.344
C00607=1045.170,-77.421,427.159,169.496,33.552,156.344
C00608=1045.176,-77.171,427.149,169.498,33.552,156.344
C00609=1045.182,-76.921,427.137,169.501,33.553,156.344
C00610=1045.188,-76.672,427.126,169.503,33.554,156.344
C00611=1045.195,-76.422,427.114,169.505,33.554,156.344
C00612=1045.200,-76.172,427.104,169.507,33.555,156.344
C00613=1045.207,-75.923,427.092,169.510,33.556,156.344
C00614=1045.213,-75.673,427.080,169.512,33.556,156.344
C00615=1045.219,-75.423,427.069,169.514,33.557,156.344
C00616=1045.226,-75.173,427.058,169.516,33.557,156.344
C00617=1045.231,-74.924,427.047,169.519,33.558,156.344
C00618=1045.238,-74.674,427.035,169.521,33.559,156.344
C00619=1045.244,-74.425,427.024,169.523,33.560,156.344
C00620=1045.250,-74.175,427.013,169.525,33.560,156.344
C00621=1045.257,-73.925,427.001,169.528,33.561,156.344
C00622=1045.263,-73.676,426.990,169.530,33.562,156.344
C00623=1045.268,-73.425,426.978,169.532,33.562,156.344
C00624=1045.274,-73.176,426.966,169.534,33.563,156.344
C00625=1045.280,-72.926,426.955,169.536,33.564,156.345
C00626=1045.287,-72.677,426.943,169.539,33.565,156.345
C00627=1045.293,-72.427,426.932,169.541,33.566,156.345
C00628=1045.299,-72.177,426.920,169.543,33.566,156.345
C00629=1045.305,-71.928,426.909,169.545,33.567,156.345
C00630=1045.311,-71.678,426.897,169.547,33.568,156.345
C00631=1045.317,-71.429,426.886,169.550,33.569,156.345
C00632=1045.323,-71.179,426.873,169.552,33.570,156.345
C00633=1045.329,-70.930,426.862,169.554,33.570,156.345
C00634=1045.335,-70.680,426.851,169.556,33.571,156.345
C00635=1045.342,-70.430,426.839,169.558,33.572,156.345
C00636=1045.347,-70.180,426.827,169.561,33.573,156.345
C00637=1045.354,-69.931,426.815,169.563,33.574,156.345
C00638=1045.360,-69.681,426.804,169.565,33.574,156.346
C00639=1045.366,-69.432,426.792,169.567,33.575,156.346
C00640=1045.372,-69.182,426.780,169.568,33.576,156.346
C00641=1045.378,-68.932,426.769,169.570,33.577,156.346
C00642=1045.384,-68.683,426.757,169.573,33.578,156.346
C00643=1045.391,-68.433,426.746,169.575,33.578,156.346
C00644=1045.396,-68.183,426.734,169.577,33.579,156.346
C00645=1045.402,-67.934,426.722,169.579,33.580,156.346
C00646=1045.409,-67.651,426.709,169.582,33.581,156.346
C00647=1045.416,-67.368,426.696,169.584,33.582,156.346
C00648=1045.423,-67.086,426.682,169.587,33.583,156.346
C00649=1045.430,-66.803,426.668,169.589,33.583,156.346
C00650=1045.436,-66.554,426.657,169.591,33.584,156.346
C00651=1045.443,-66.305,426.645,169.593,33.585,156.346
C00652=1045.449,-66.054,426.633,169.596,33.586,156.347
C00653=1045.455,-65.805,426.622,169.598,33.587,156.347
C00654=1045.461,-65.556,426.610,169.600,33.588,156.347
C00655=1045.467,-65.306,426.597,169.602,33.589,156.347
C00656=1045.474,-65.056,426.586,169.604,33.590,156.347
C00657=1045.480,-64.807,426.574,169.607,33.591,156.347
C00658=1045.486,-64.557,426.562,169.609,33.591,156.347
C00659=1045.492,-64.307,426.550,169.611,33.592,156.347
C00660=1045.498,-64.058,426.539,169.613,33.593,156.347
C00661=1045.505,-63.808,426.527,169.615,33.594,156.347
C00662=1045.510,-63.558,426.514,169.617,33.594,156.347
C00663=1045.517,-63.309,426.502,169.620,33.595,156.347
C00664=1045.523,-63.059,426.491,169.622,33.596,156.347
C00665=1045.529,-62.809,426.479,169.624,33.597,156.348
C00666=1045.535,-62.560,426.467,169.626,33.598,156.348
C00667=1045.542,-62.310,426.455,169.628,33.598,156.348
C00668=1045.548,-62.060,426.442,169.630,33.600,156.348
C00669=1045.554,-61.811,426.431,169.633,33.601,156.348
C00670=1045.560,-61.561,426.420,169.635,33.602,156.348
C00671=1045.566,-61.311,426.407,169.637,33.602,156.348
C00672=1045.573,-61.062,426.395,169.639,33.603,156.348
C00673=1045.580,-60.812,426.383,169.641,33.604,156.348
C00674=1045.585,-60.562,426.371,169.643,33.605,156.348
C00675=1045.592,-60.313,426.359,169.646,33.606,156.348
C00676=1045.598,-60.064,426.347,169.648,33.606,156.348
C00677=1045.604,-59.814,426.334,169.650,33.608,156.349
C00678=1045.610,-59.564,426.323,169.652,33.609,156.349
C00679=1045.617,-59.314,426.311,169.654,33.609,156.349
C00680=1045.623,-59.064,426.299,169.656,33.610,156.349
C00681=1045.629,-58.815,426.287,169.659,33.611,156.349
C00682=1045.636,-58.566,426.275,169.661,33.612,156.349
C00683=1045.642,-58.316,426.263,169.663,33.613,156.349
C00684=1045.648,-58.066,426.251,169.665,33.613,156.349
C00685=1045.655,-57.817,426.239,169.667,33.615,156.349
C00686=1045.661,-57.567,426.226,169.669,33.616,156.349
C00687=1045.667,-57.317,426.214,169.671,33.616,156.350
C00688=1045.673,-57.068,426.202,169.674,33.617,156.350
C00689=1045.680,-56.818,426.190,169.676,33.618,156.350
C00690=1045.687,-56.568,426.178,169.678,33.619,156.350
C00691=1045.692,-56.319,426.165,169.680,33.620,156.350
C00692=1045.699,-56.070,426.154,169.682,33.621,156.350
C00693=1045.705,-55.820,426.142,169.684,33.622,156.350
C00694=1045.711,-55.570,426.129,169.686,33.623,156.350
C00695=1045.718,-55.321,426.117,169.689,33.623,156.350
C00696=1045.724,-55.071,426.104,169.691,33.624,156.350
C00697=1045.730,-54.821,426.093,169.693,33.625,156.350
C00698=1045.737,-54.572,426.081,169.695,33.626,156.351
C00699=1045.743,-54.322,426.068,169.697,33.627,156.351
C00700=1045.750,-54.073,426.055,169.699,33.628,156.351
C00701=1045.756,-53.823,426.043,169.701,33.629,156.351
C00702=1045.762,-53.573,426.031,169.704,33.630,156.351
C00703=1045.769,-53.324,426.019,169.706,33.630,156.351
C00704=1045.775,-53.074,426.006,169.708,33.632,156.351
C00705=1045.782,-52.824,425.994,169.710,33.633,156.351
C00706=1045.788,-52.574,425.982,169.712,33.633,156.351
C00707=1045.794,-52.325,425.970,169.714,33.634,156.351
C00708=1045.801,-52.076,425.957,169.716,33.635,156.351
C00709=1045.807,-51.826,425.945,169.719,33.637,156.352
C00710=1045.813,-51.545,425.931,169.721,33.637,156.352
C00711=1045.822,-51.264,425.917,169.723,33.638,156.352
C00712=1045.829,-50.982,425.903,169.726,33.640,156.352
C00713=1045.836,-50.701,425.889,169.728,33.640,156.352
C00714=1045.842,-50.452,425.877,169.730,33.641,156.352
C00715=1045.848,-50.202,425.864,169.732,33.643,156.352
C00716=1045.854,-49.952,425.852,169.734,33.643,156.352
C00717=1045.861,-49.703,425.839,169.737,33.645,156.353
C00718=1045.867,-49.453,425.827,169.738,33.646,156.353
C00719=1045.873,-49.203,425.814,169.740,33.646,156.353
C00720=1045.879,-48.954,425.801,169.742,33.648,156.353
C00721=1045.886,-48.705,425.789,169.744,33.649,156.353
C00722=1045.892,-48.455,425.776,169.746,33.650,156.353
C00723=1045.898,-48.205,425.763,169.748,33.651,156.353
C00724=1045.904,-47.955,425.750,169.750,33.652,156.353
C00725=1045.910,-47.706,425.739,169.752,33.653,156.353
C00726=1045.917,-47.457,425.725,169.754,33.654,156.354
C00727=1045.923,-47.207,425.713,169.756,33.655,156.354
C00728=1045.928,-46.957,425.700,169.758,33.656,156.354
C00729=1045.935,-46.708,425.687,169.760,33.657,156.354
C00730=1045.941,-46.458,425.675,169.763,33.658,156.354
C00731=1045.947,-46.208,425.662,169.765,33.660,156.354
C00732=1045.953,-45.959,425.649,169.767,33.660,156.354
C00733=1045.959,-45.709,425.637,169.769,33.662,156.355
C00734=1045.967,-45.459,425.623,169.771,33.663,156.355
C00735=1045.973,-45.209,425.611,169.773,33.664,156.355
C00736=1045.979,-44.960,425.598,169.775,33.665,156.355
C00737=1045.985,-44.710,425.585,169.777,33.666,156.355
C00738=1045.992,-44.461,425.573,169.779,33.667,156.355
C00739=1045.998,-44.212,425.560,169.781,33.668,156.355
C00740=1046.004,-43.962,425.547,169.783,33.669,156.355
C00741=1046.010,-43.712,425.534,169.785,33.671,156.356
C00742=1046.016,-43.462,425.522,169.787,33.671,156.356
C00743=1046.023,-43.214,425.509,169.789,33.673,156.356
C00744=1046.029,-42.964,425.496,169.792,33.674,156.356
C00745=1046.036,-42.714,425.483,169.794,33.675,156.356
C00746=1046.041,-42.464,425.470,169.796,33.676,156.356
C00747=1046.048,-42.215,425.457,169.798,33.677,156.356
C00748=1046.054,-41.965,425.445,169.800,33.678,156.356
C00749=1046.061,-41.716,425.432,169.802,33.680,156.357
C00750=1046.067,-41.466,425.418,169.804,33.680,156.357
C00751=1046.073,-41.217,425.406,169.806,33.682,156.357
C00752=1046.079,-40.967,425.392,169.808,33.682,156.357
C00753=1046.086,-40.717,425.380,169.810,33.684,156.357
C00754=1046.092,-40.468,425.367,169.812,33.685,156.357
C00755=1046.098,-40.218,425.354,169.814,33.686,156.357
C00756=1046.104,-39.969,425.341,169.816,33.687,156.358
C00757=1046.111,-39.719,425.328,169.818,33.688,156.358
C00758=1046.117,-39.469,425.315,169.820,33.689,156.358
C00759=1046.124,-39.220,425.302,169.822,33.690,156.358
C00760=1046.130,-38.970,425.290,169.824,33.691,156.358
C00761=1046.136,-38.721,425.276,169.826,33.693,156.358
C00762=1046.142,-38.471,425.263,169.828,33.693,156.358
C00763=1046.149,-38.221,425.250,169.831,33.695,156.359
C00764=1046.155,-37.972,425.237,169.833,33.696,156.359
C00765=1046.161,-37.722,425.224,169.835,33.697,156.359
C00766=1046.168,-37.473,425.210,169.837,33.699,156.359
C00767=1046.173,-37.223,425.198,169.839,33.700,156.359
C00768=1046.180,-36.974,425.185,169.841,33.701,156.359
C00769=1046.186,-36.724,425.170,169.843,33.702,156.359
C00770=1046.192,-36.474,425.158,169.845,33.704,156.360
C00771=1046.198,-36.224,425.145,169.847,33.704,156.360
C00772=1046.204,-35.975,425.131,169.849,33.706,156.360
C00773=1046.210,-35.726,425.118,169.851,33.707,156.360
C00774=1046.218,-35.444,425.104,169.853,33.709,156.360
C00775=1046.225,-35.164,425.089,169.855,33.710,156.361
C00776=1046.232,-34.883,425.073,169.857,33.711,156.361
C00777=1046.238,-34.603,425.059,169.860,33.712,156.361
C00778=1046.245,-34.353,425.046,169.862,33.714,156.361
C00779=1046.251,-34.103,425.032,169.864,33.715,156.361
C00780=1046.258,-33.854,425.019,169.866,33.716,156.361
C00781=1046.264,-33.605,425.006,169.868,33.717,156.361
C00782=1046.270,-33.356,424.992,169.870,33.719,156.362
C00783=1046.277,-33.105,424.979,169.872,33.720,156.362
C00784=1046.282,-32.855,424.965,169.874,33.721,156.362
C00785=1046.288,-32.606,424.952,169.876,33.722,156.362
C00786=1046.295,-32.356,424.939,169.878,33.724,156.362
C00787=1046.301,-32.107,424.925,169.880,33.724,156.362
C00788=1046.308,-31.858,424.912,169.882,33.726,156.363
C00789=1046.314,-31.608,424.899,169.884,33.727,156.363
C00790=1046.321,-31.358,424.885,169.886,33.729,156.363
C00791=1046.327,-31.109,424.872,169.888,33.729,156.363
C00792=1046.333,-30.859,424.859,169.890,33.731,156.363
C00793=1046.340,-30.609,424.846,169.892,33.732,156.363
C00794=1046.345,-30.360,424.832,169.894,33.733,156.363
C00795=1046.351,-30.110,424.819,169.896,33.734,156.364
C00796=1046.358,-29.861,424.805,169.898,33.736,156.364
C00797=1046.364,-29.611,424.792,169.900,33.737,156.364
C00798=1046.370,-29.362,424.778,169.902,33.738,156.364
C00799=1046.377,-29.112,424.765,169.904,33.739,156.364
C00800=1046.383,-28.863,424.751,169.906,33.741,156.365
C00801=1046.390,-28.614,424.738,169.908,33.742,156.365
C00802=1046.396,-28.363,424.724,169.910,33.743,156.365
C00803=1046.402,-28.114,424.711,169.912,33.744,156.365
C00804=1046.408,-27.865,424.697,169.914,33.746,156.365
C00805=1046.415,-27.615,424.684,169.916,33.747,156.365
C00806=1046.421,-27.365,424.671,169.918,33.748,156.365
C00807=1046.428,-27.115,424.657,169.920,33.749,156.366
C00808=1046.434,-26.866,424.644,169.922,33.751,156.366
C00809=1046.440,-26.617,424.630,169.923,33.752,156.366
C00810=1046.447,-26.367,424.616,169.925,33.754,156.366
C00811=1046.452,-26.118,424.602,169.927,33.754,156.366
C00812=1046.459,-25.868,424.588,169.929,33.756,156.367
C00813=1046.465,-25.619,424.575,169.931,33.757,156.367
C00814=1046.471,-25.369,424.561,169.934,33.758,156.367
C00815=1046.477,-25.120,424.547,169.936,33.760,156.367
C00816=1046.484,-24.870,424.534,169.938,33.761,156.367
C00817=1046.489,-24.620,424.520,169.940,33.763,156.367
C00818=1046.496,-24.371,424.506,169.942,33.764,156.368
C00819=1046.503,-24.122,424.492,169.944,33.766,156.368
C00820=1046.508,-23.872,424.479,169.946,33.767,156.368
C00821=1046.515,-23.622,424.465,169.948,33.768,156.368
C00822=1046.520,-23.372,424.451,169.950,33.769,156.368
C00823=1046.528,-23.123,424.437,169.952,33.770,156.369
C00824=1046.534,-22.874,424.423,169.954,33.772,156.369
C00825=1046.539,-22.624,424.410,169.956,33.773,156.369
C00826=1046.546,-22.374,424.396,169.958,33.775,156.369
C00827=1046.552,-22.125,424.382,169.960,33.776,156.369
C00828=1046.559,-21.875,424.368,169.961,33.777,156.369
C00829=1046.565,-21.626,424.354,169.963,33.779,156.370
C00830=1046.571,-21.376,424.340,169.965,33.780,156.370
C00831=1046.577,-21.127,424.327,169.967,33.782,156.370
C00832=1046.584,-20.877,424.313,169.969,33.782,156.370
C00833=1046.590,-20.628,424.299,169.971,33.784,156.370
C00834=1046.596,-20.378,424.285,169.973,33.785,156.371
C00835=1046.602,-20.129,424.270,169.975,33.787,156.371
C00836=1046.609,-19.879,424.257,169.977,33.788,156.371
C00837=1046.615,-19.629,424.243,169.979,33.789,156.371
C00838=1046.622,-19.348,424.227,169.981,33.791,156.371
C00839=1046.630,-19.067,424.212,169.983,33.792,156.372
C00840=1046.637,-18.785,424.196,169.985,33.794,156.372
C00841=1046.644,-18.503,424.181,169.988,33.796,156.372
C00842=1046.650,-18.254,424.166,169.989,33.797,156.372
C00843=1046.657,-18.004,424.152,169.991,33.798,156.372
C00844=1046.662,-17.754,424.139,169.993,33.800,156.373
C00845=1046.669,-17.505,424.124,169.995,33.801,156.373
C00846=1046.675,-17.256,424.110,169.997,33.802,156.373
C00847=1046.682,-17.006,424.096,169.999,33.803,156.373
C00848=1046.688,-16.757,424.083,170.001,33.805,156.373
C00849=1046.694,-16.507,424.068,170.003,33.806,156.373
C00850=1046.701,-16.258,424.054,170.005,33.808,156.374
C00851=1046.707,-16.008,424.040,170.007,33.809,156.374
C00852=1046.713,-15.759,424.026,170.009,33.810,156.374
C00853=1046.719,-15.509,424.012,170.011,33.812,156.374
C00854=1046.726,-15.259,423.998,170.012,33.813,156.374
C00855=1046.732,-15.010,423.984,170.014,33.815,156.375
C00856=1046.739,-14.761,423.969,170.016,33.816,156.375
C00857=1046.744,-14.511,423.956,170.018,33.817,156.375
C00858=1046.751,-14.261,423.941,170.020,33.819,156.375
C00859=1046.757,-14.012,423.927,170.022,33.820,156.375
C00860=1046.763,-13.762,423.912,170.024,33.821,156.376
C00861=1046.769,-13.513,423.899,170.026,33.823,156.376
C00862=1046.776,-13.263,423.884,170.028,33.825,156.376
C00863=1046.782,-13.014,423.870,170.029,33.826,156.376
C00864=1046.788,-12.764,423.855,170.031,33.828,156.377
C00865=1046.795,-12.514,423.842,170.033,33.829,156.377
C00866=1046.801,-12.265,423.827,170.035,33.830,156.377
C00867=1046.807,-12.016,423.812,170.037,33.832,156.377
C00868=1046.813,-11.766,423.799,170.039,33.833,156.377
C00869=1046.820,-11.517,423.784,170.041,33.835,156.377
C00870=1046.825,-11.267,423.770,170.043,33.836,156.378
C00871=1046.831,-11.018,423.755,170.045,33.837,156.378
C00872=1046.838,-10.768,423.741,170.046,33.839,156.378
C00873=1046.844,-10.519,423.727,170.048,33.840,156.378
C00874=1046.850,-10.269,423.712,170.050,33.842,156.379
C00875=1046.857,-10.020,423.698,170.052,33.844,156.379
C00876=1046.863,-9.770,423.684,170.054,33.845,156.379
C00877=1046.869,-9.520,423.669,170.056,33.846,156.379
C00878=1046.876,-9.272,423.655,170.058,33.848,156.379
C00879=1046.882,-9.021,423.641,170.059,33.849,156.380
C00880=1046.888,-8.772,423.626,170.061,33.850,156.380
C00881=1046.894,-8.523,423.611,170.063,33.852,156.380
C00882=1046.901,-8.273,423.598,170.065,33.853,156.380
C00883=1046.907,-8.023,423.583,170.067,33.855,156.380
C00884=1046.913,-7.774,423.568,170.069,33.857,156.381
C00885=1046.920,-7.525,423.554,170.071,33.858,156.381
C00886=1046.926,-7.275,423.539,170.073,33.859,156.381
C00887=1046.932,-7.026,423.525,170.074,33.861,156.381
C00888=1046.938,-6.776,423.510,170.077,33.862,156.381
C00889=1046.946,-6.527,423.496,170.079,33.864,156.382
C00890=1046.951,-6.277,423.482,170.081,33.865,156.382
C00891=1046.957,-6.027,423.467,170.083,33.866,156.382
C00892=1046.965,-5.778,423.452,170.085,33.868,156.382
C00893=1046.971,-5.528,423.437,170.087,33.869,156.382
C00894=1046.976,-5.279,423.424,170.088,33.871,156.383
C00895=1046.983,-5.029,423.409,170.090,33.872,156.383
C00896=1046.990,-4.780,423.394,170.092,33.874,156.383
C00897=1046.996,-4.531,423.380,170.094,33.875,156.383
C00898=1047.002,-4.281,423.365,170.096,33.877,156.384
C00899=1047.008,-4.032,423.350,170.098,33.878,156.384
C00900=1047.015,-3.782,423.336,170.100,33.879,156.384
C00901=1047.021,-3.533,423.322,170.101,33.881,156.384
C00902=1047.028,-3.250,423.304,170.103,33.883,156.384
C00903=1047.036,-2.966,423.288,170.106,33.884,156.385
C00904=1047.042,-2.683,423.270,170.108,33.886,156.385
C00905=1047.049,-2.400,423.254,170.110,33.888,156.385
C00906=1047.055,-2.151,423.240,170.112,33.890,156.385
C00907=1047.061,-1.901,423.225,170.113,33.891,156.386
C00908=1047.068,-1.651,423.210,170.115,33.893,156.386
C00909=1047.074,-1.402,423.195,170.117,33.894,156.386
C00910=1047.080,-1.153,423.180,170.119,33.896,156.386
C00911=1047.086,-0.903,423.165,170.121,33.897,156.387
C00912=1047.093,-0.654,423.150,170.122,33.899,156.387
C00913=1047.098,-0.405,423.136,170.124,33.900,156.387
C00914=1047.105,-0.155,423.121,170.126,33.902,156.387
C00915=1047.111,0.095,423.106,170.128,33.904,156.388
C00916=1047.118,0.344,423.091,170.130,33.905,156.388
C00917=1047.123,0.593,423.076,170.131,33.907,156.388
C00918=1047.129,0.843,423.061,170.133,33.909,156.388
C00919=1047.135,1.093,423.046,170.135,33.910,156.389
C00920=1047.142,1.343,423.031,170.137,33.911,156.389
C00921=1047.148,1.592,423.016,170.139,33.913,156.389
C00922=1047.154,1.841,423.001,170.140,33.915,156.389
C00923=1047.160,2.091,422.986,170.142,33.916,156.389
C00924=1047.167,2.340,422.971,170.144,33.917,156.390
C00925=1047.173,2.590,422.956,170.146,33.919,156.390
C00926=1047.179,2.839,422.941,170.148,33.921,156.390
C00927=1047.186,3.088,422.926,170.149,33.922,156.390
C00928=1047.192,3.338,422.911,170.151,33.924,156.391
C00929=1047.198,3.588,422.896,170.153,33.926,156.391
C00930=1047.205,3.837,422.881,170.155,33.927,156.391
C00931=1047.211,4.086,422.867,170.158,33.928,156.391
C00932=1047.216,4.336,422.851,170.159,33.930,156.392
C00933=1047.223,4.585,422.836,170.161,33.932,156.392
C00934=1047.229,4.835,422.821,170.163,33.933,156.392
C00935=1047.236,5.084,422.806,170.165,33.935,156.392
C00936=1047.242,5.334,422.791,170.167,33.936,156.392
C00937=1047.248,5.583,422.776,170.168,33.938,156.393
C00938=1047.254,5.833,422.761,170.170,33.939,156.393
C00939=1047.261,6.082,422.746,170.172,33.941,156.393
C00940=1047.267,6.331,422.731,170.174,33.943,156.393
C00941=1047.274,6.581,422.716,170.176,33.944,156.394
C00942=1047.279,6.831,422.700,170.177,33.946,156.394
C00943=1047.286,7.080,422.684,170.179,33.947,156.394
C00944=1047.292,7.329,422.670,170.181,33.949,156.394
C00945=1047.298,7.579,422.655,170.183,33.951,156.395
C00946=1047.305,7.828,422.640,170.185,33.952,156.395
C00947=1047.311,8.077,422.624,170.186,33.953,156.395
C00948=1047.318,8.327,422.609,170.188,33.955,156.395
C00949=1047.324,8.577,422.594,170.190,33.957,156.396
C00950=1047.330,8.826,422.579,170.192,33.958,156.396
C00951=1047.336,9.076,422.563,170.194,33.960,156.396
C00952=1047.343,9.325,422.548,170.195,33.961,156.396
C00953=1047.349,9.575,422.533,170.197,33.963,156.396
C00954=1047.356,9.824,422.518,170.199,33.964,156.397
C00955=1047.362,10.073,422.503,170.201,33.966,156.397
C00956=1047.368,10.323,422.488,170.202,33.968,156.397
C00957=1047.375,10.572,422.472,170.204,33.969,156.397
C00958=1047.380,10.822,422.457,170.206,33.970,156.398
C00959=1047.387,11.071,422.442,170.208,33.972,156.398
C00960=1047.393,11.320,422.426,170.210,33.974,156.398
C00961=1047.400,11.570,422.411,170.211,33.975,156.398
C00962=1047.406,11.820,422.396,170.213,33.977,156.399
C00963=1047.413,12.069,422.381,170.215,33.978,156.399
C00964=1047.419,12.318,422.366,170.217,33.980,156.399
C00965=1047.425,12.568,422.350,170.219,33.982,156.399
C00966=1047.432,12.854,422.333,170.221,33.983,156.400
C00967=1047.439,13.138,422.315,170.223,33.985,156.400
C00968=1047.447,13.423,422.298,170.226,33.987,156.400
C00969=1047.454,13.709,422.280,170.228,33.989,156.400
C00970=1047.461,13.958,422.264,170.229,33.990,156.401
C00971=1047.467,14.207,422.249,170.231,33.992,156.401
C00972=1047.474,14.456,422.234,170.233,33.993,156.401
C00973=1047.480,14.706,422.218,170.235,33.995,156.401
C00974=1047.486,14.955,422.202,170.236,33.997,156.402
C00975=1047.492,15.205,422.187,170.238,33.998,156.402
C00976=1047.499,15.454,422.171,170.240,34.000,156.402
C00977=1047.505,15.704,422.156,170.242,34.001,156.402
C00978=1047.511,15.953,422.140,170.243,34.003,156.403
C00979=1047.518,16.203,422.125,170.245,34.005,156.403
C00980=1047.523,16.452,422.109,170.247,34.007,156.403
C00981=1047.530,16.702,422.094,170.249,34.008,156.403
C00982=1047.537,16.951,422.078,170.250,34.009,156.404
C00983=1047.542,17.201,422.063,170.252,34.011,156.404
C00984=1047.549,17.450,422.047,170.254,34.013,156.404
C00985=1047.555,17.699,422.031,170.256,34.015,156.404
C00986=1047.561,17.949,422.016,170.257,34.016,156.405
C00987=1047.568,18.198,422.000,170.259,34.018,156.405
C00988=1047.574,18.448,421.985,170.261,34.019,156.405
C00989=1047.580,18.697,421.969,170.262,34.021,156.405
C00990=1047.586,18.946,421.953,170.264,34.023,156.406
C00991=1047.593,19.196,421.938,170.266,34.024,156.406
C00992=1047.599,19.445,421.922,170.268,34.026,156.406
C00993=1047.605,19.694,421.906,170.269,34.027,156.406
C00994=1047.612,19.944,421.891,170.272,34.029,156.407
C00995=1047.618,20.193,421.875,170.274,34.031,156.407
C00996=1047.624,20.442,421.859,170.276,34.033,156.407
C00997=1047.630,20.692,421.843,170.277,34.034,156.407
C00998=1047.637,20.941,421.828,170.279,34.036,156.408
C00999=1047.643,21.191,421.812,170.281,34.037,156.408
C01000=1047.648,21.441,421.796,170.283,34.039,156.408
C01001=1047.655,21.691,421.780,170.284,34.041,156.408
C01002=1047.661,21.940,421.764,170.286,34.043,156.409
C01003=1047.668,22.189,421.748,170.288,34.044,156.409
C01004=1047.674,22.439,421.733,170.289,34.046,156.409
C01005=1047.680,22.688,421.717,170.291,34.047,156.410
C01006=1047.686,22.937,421.701,170.293,34.049,156.410
C01007=1047.693,23.186,421.685,170.295,34.051,156.410
C01008=1047.699,23.436,421.669,170.296,34.053,156.410
C01009=1047.705,23.686,421.653,170.298,34.054,156.411
C01010=1047.711,23.935,421.637,170.300,34.056,156.411
C01011=1047.717,24.184,421.621,170.301,34.057,156.411
C01012=1047.725,24.434,421.605,170.303,34.059,156.411
C01013=1047.731,24.683,421.589,170.305,34.061,156.412
C01014=1047.737,24.933,421.574,170.307,34.063,156.412
C01015=1047.743,25.182,421.558,170.308,34.064,156.412
C01016=1047.749,25.431,421.541,170.310,34.066,156.412
C01017=1047.756,25.680,421.526,170.312,34.068,156.413
C01018=1047.761,25.930,421.510,170.313,34.069,156.413
C01019=1047.769,26.180,421.494,170.315,34.071,156.413
C01020=1047.774,26.430,421.478,170.318,34.072,156.413
C01021=1047.780,26.679,421.462,170.320,34.074,156.414
C01022=1047.787,26.928,421.446,170.321,34.075,156.414
C01023=1047.793,27.177,421.430,170.323,34.077,156.414
C01024=1047.800,27.426,421.414,170.325,34.079,156.415
C01025=1047.806,27.676,421.398,170.326,34.081,156.415
C01026=1047.812,27.926,421.381,170.328,34.083,156.415
C01027=1047.819,28.175,421.366,170.330,34.084,156.415
C01028=1047.825,28.424,421.349,170.332,34.086,156.416
C01029=1047.831,28.673,421.333,170.333,34.087,156.416
C01030=1047.838,28.960,421.314,170.335,34.089,156.416
C01031=1047.845,29.247,421.297,170.337,34.091,156.416
C01032=1047.853,29.533,421.278,170.339,34.093,156.417
C01033=1047.859,29.819,421.259,170.341,34.095,156.417
C01034=1047.866,30.068,421.243,170.343,34.097,156.417
C01035=1047.872,30.318,421.227,170.344,34.099,156.418
C01036=1047.878,30.567,421.210,170.346,34.101,156.418
C01037=1047.884,30.816,421.194,170.348,34.102,156.418
C01038=1047.890,31.066,421.178,170.349,34.104,156.418
C01039=1047.897,31.315,421.162,170.351,34.106,156.419
C01040=1047.903,31.565,421.146,170.353,34.107,156.419
C01041=1047.909,31.814,421.129,170.355,34.109,156.419
C01042=1047.915,32.064,421.113,170.356,34.111,156.419
C01043=1047.922,32.313,421.096,170.359,34.113,156.420
C01044=1047.929,32.562,421.080,170.361,34.115,156.420
C01045=1047.934,32.811,421.064,170.362,34.116,156.420
C01046=1047.940,33.061,421.048,170.364,34.118,156.421
C01047=1047.947,33.311,421.031,170.366,34.119,156.421
C01048=1047.953,33.560,421.015,170.367,34.121,156.421
C01049=1047.960,33.809,420.999,170.369,34.123,156.421
C01050=1047.966,34.058,420.983,170.371,34.125,156.422
C01051=1047.972,34.307,420.966,170.372,34.127,156.422
C01052=1047.978,34.557,420.949,170.374,34.128,156.422
C01053=1047.984,34.807,420.933,170.376,34.130,156.423
C01054=1047.990,35.056,420.917,170.377,34.131,156.423
C01055=1047.998,35.306,420.901,170.379,34.133,156.423
C01056=1048.004,35.555,420.884,170.381,34.135,156.423
C01057=1048.010,35.804,420.867,170.382,34.136,156.424
C01058=1048.016,36.053,420.851,170.384,34.138,156.424
C01059=1048.022,36.303,420.835,170.386,34.140,156.424
C01060=1048.028,36.553,420.818,170.388,34.142,156.424
C01061=1048.034,36.802,420.802,170.389,34.143,156.425
C01062=1048.042,37.051,420.785,170.391,34.145,156.425
C01063=1048.048,37.300,420.769,170.393,34.147,156.425
C01064=1048.054,37.550,420.753,170.395,34.148,156.426
C01065=1048.060,37.800,420.736,170.397,34.150,156.426
C01066=1048.066,38.048,420.719,170.399,34.152,156.426
C01067=1048.072,38.298,420.703,170.400,34.154,156.426
C01068=1048.078,38.547,420.687,170.402,34.156,156.427
C01069=1048.085,38.797,420.669,170.404,34.157,156.427
C01070=1048.091,39.046,420.653,170.405,34.159,156.427
C01071=1048.097,39.295,420.637,170.407,34.161,156.428
C01072=1048.104,39.545,420.620,170.409,34.163,156.428
C01073=1048.110,39.794,420.603,170.410,34.164,156.428
C01074=1048.115,40.044,420.586,170.412,34.166,156.428
C01075=1048.121,40.292,420.569,170.414,34.168,156.429
C01076=1048.128,40.543,420.553,170.415,34.170,156.429
C01077=1048.134,40.792,420.537,170.417,34.172,156.429
C01078=1048.140,41.041,420.520,170.419,34.173,156.430
C01079=1048.147,41.291,420.503,170.420,34.175,156.430
C01080=1048.153,41.540,420.487,170.422,34.177,156.430
C01081=1048.159,41.789,420.470,170.424,34.179,156.430
C01082=1048.165,42.039,420.453,170.425,34.180,156.431
C01083=1048.172,42.287,420.436,170.428,34.182,156.431
C01084=1048.178,42.537,420.420,170.430,34.184,156.431
C01085=1048.185,42.786,420.403,170.431,34.185,156.431
C01086=1048.191,43.036,420.386,170.433,34.187,156.432
C01087=1048.197,43.286,420.370,170.435,34.189,156.432
C01088=1048.203,43.535,420.352,170.436,34.191,156.432
C01089=1048.209,43.784,420.336,170.438,34.193,156.433
C01090=1048.215,44.033,420.319,170.439,34.194,156.433
C01091=1048.221,44.283,420.302,170.441,34.196,156.433
C01092=1048.227,44.532,420.285,170.443,34.198,156.434
C01093=1048.233,44.782,420.268,170.444,34.200,156.434
C01094=1048.240,45.068,420.248,170.446,34.202,156.434
C01095=1048.247,45.354,420.229,170.448,34.204,156.435
C01096=1048.255,45.640,420.210,170.450,34.206,156.435
C01097=1048.261,45.927,420.190,170.452,34.208,156.435
C01098=1048.267,46.176,420.173,170.454,34.210,156.436
C01099=1048.273,46.426,420.156,170.455,34.212,156.436
C01100=1048.280,46.674,420.139,170.457,34.214,156.436
C01101=1048.285,46.923,420.122,170.459,34.215,156.436
C01102=1048.292,47.174,420.105,170.461,34.217,156.437
C01103=1048.298,47.422,420.088,170.463,34.219,156.437
C01104=1048.304,47.673,420.071,170.464,34.221,156.437
C01105=1048.310,47.921,420.054,170.466,34.223,156.438
C01106=1048.316,48.170,420.037,170.468,34.225,156.438
C01107=1048.322,48.420,420.020,170.469,34.227,156.438
C01108=1048.328,48.669,420.003,170.471,34.229,156.439
C01109=1048.335,48.919,419.985,170.473,34.230,156.439
C01110=1048.341,49.168,419.968,170.474,34.232,156.439
C01111=1048.347,49.417,419.951,170.476,34.234,156.439
C01112=1048.354,49.666,419.934,170.477,34.236,156.440
C01113=1048.359,49.916,419.917,170.479,34.237,156.440
C01114=1048.366,50.165,419.900,170.481,34.239,156.440
C01115=1048.372,50.414,419.883,170.482,34.241,156.441
C01116=1048.378,50.665,419.866,170.484,34.243,156.441
C01117=1048.384,50.913,419.849,170.486,34.245,156.441
C01118=1048.391,51.163,419.831,170.488,34.246,156.441
C01119=1048.396,51.412,419.815,170.490,34.248,156.442
C01120=1048.402,51.661,419.798,170.492,34.250,156.442
C01121=1048.409,51.911,419.780,170.493,34.252,156.442
C01122=1048.415,52.160,419.763,170.495,34.254,156.443
C01123=1048.421,52.410,419.746,170.496,34.255,156.443
C01124=1048.428,52.658,419.729,170.498,34.257,156.443
C01125=1048.434,52.908,419.711,170.500,34.259,156.444
C01126=1048.440,53.157,419.694,170.501,34.261,156.444
C01127=1048.446,53.407,419.676,170.503,34.263,156.444
C01128=1048.452,53.656,419.660,170.505,34.265,156.444
C01129=1048.459,53.905,419.643,170.506,34.267,156.445
C01130=1048.464,54.154,419.625,170.508,34.268,156.445
C01131=1048.471,54.404,419.608,170.510,34.270,156.445
C01132=1048.477,54.653,419.591,170.511,34.272,156.446
C01133=1048.483,54.903,419.574,170.513,34.274,156.446
C01134=1048.490,55.152,419.557,170.514,34.275,156.446
C01135=1048.496,55.401,419.539,170.517,34.277,156.447
C01136=1048.503,55.651,419.521,170.519,34.279,156.447
C01137=1048.509,55.900,419.504,170.520,34.280,156.447
C01138=1048.515,56.149,419.486,170.522,34.282,156.447
C01139=1048.521,56.398,419.469,170.524,34.284,156.448
C01140=1048.527,56.648,419.452,170.525,34.286,156.448
C01141=1048.533,56.897,419.435,170.527,34.288,156.448
C01142=1048.540,57.147,419.418,170.529,34.290,156.449
C01143=1048.546,57.396,419.400,170.530,34.291,156.449
C01144=1048.552,57.645,419.383,170.532,34.293,156.449
C01145=1048.559,57.895,419.365,170.533,34.295,156.449
C01146=1048.565,58.143,419.348,170.535,34.297,156.450
C01147=1048.572,58.393,419.331,170.537,34.299,156.450
C01148=1048.577,58.642,419.313,170.538,34.300,156.450
C01149=1048.584,58.891,419.296,170.540,34.302,156.451
C01150=1048.590,59.141,419.278,170.542,34.304,156.451
C01151=1048.596,59.390,419.261,170.544,34.306,156.451
C01152=1048.603,59.640,419.243,170.546,34.307,156.451
C01153=1048.609,59.888,419.226,170.548,34.309,156.452
C01154=1048.616,60.138,419.209,170.549,34.311,156.452
C01155=1048.622,60.387,419.191,170.551,34.312,156.452
C01156=1048.628,60.636,419.174,170.553,34.314,156.453
C01157=1048.634,60.886,419.156,170.554,34.316,156.453
C01158=1048.641,61.172,419.136,170.556,34.318,156.453
C01159=1048.649,61.458,419.116,170.558,34.320,156.454
C01160=1048.656,61.744,419.096,170.560,34.322,156.454
C01161=1048.663,62.030,419.076,170.562,34.324,156.454
C01162=1048.670,62.280,419.059,170.563,34.326,156.455
C01163=1048.676,62.529,419.041,170.565,34.328,156.455
C01164=1048.683,62.778,419.024,170.567,34.329,156.455
C01165=1048.689,63.027,419.005,170.568,34.331,156.455
C01166=1048.695,63.276,418.988,170.571,34.333,156.456
C01167=1048.701,63.526,418.971,170.573,34.335,156.456
C01168=1048.708,63.775,418.953,170.574,34.337,156.456
C01169=1048.714,64.024,418.936,170.576,34.339,156.457
C01170=1048.721,64.273,418.918,170.578,34.340,156.457
C01171=1048.727,64.523,418.900,170.579,34.342,156.457
C01172=1048.733,64.773,418.882,170.581,34.344,156.458
C01173=1048.739,65.022,418.865,170.582,34.346,156.458
C01174=1048.746,65.271,418.847,170.584,34.348,156.458
C01175=1048.752,65.521,418.829,170.586,34.350,156.459
C01176=1048.758,65.769,418.812,170.587,34.351,156.459
C01177=1048.764,66.019,418.794,170.589,34.353,156.459
C01178=1048.770,66.269,418.776,170.591,34.355,156.459
C01179=1048.776,66.517,418.758,170.592,34.357,156.460
C01180=1048.783,66.767,418.740,170.594,34.359,156.460
C01181=1048.789,67.016,418.722,170.596,34.361,156.460
C01182=1048.795,67.265,418.705,170.598,34.362,156.461
C01183=1048.802,67.514,418.687,170.600,34.364,156.461
C01184=1048.808,67.764,418.669,170.601,34.366,156.461
C01185=1048.813,68.013,418.651,170.603,34.368,156.462
C01186=1048.819,68.263,418.633,170.605,34.370,156.462
C01187=1048.826,68.512,418.615,170.606,34.372,156.462
C01188=1048.832,68.761,418.598,170.608,34.373,156.462
C01189=1048.838,69.010,418.580,170.609,34.375,156.463
C01190=1048.845,69.259,418.561,170.611,34.377,156.463
C01191=1048.851,69.509,418.543,170.613,34.379,156.463
C01192=1048.857,69.758,418.526,170.614,34.381,156.464
C01193=1048.863,70.007,418.508,170.616,34.383,156.464
C01194=1048.870,70.257,418.490,170.618,34.384,156.464
C01195=1048.875,70.506,418.472,170.619,34.386,156.465
C01196=1048.882,70.755,418.454,170.622,34.388,156.465
C01197=1048.888,71.005,418.436,170.623,34.390,156.465
C01198=1048.894,71.254,418.417,170.625,34.392,156.466
C01199=1048.900,71.503,418.399,170.627,34.394,156.466
C01200=1048.906,71.752,418.382,170.628,34.396,156.466
C01201=1048.913,72.001,418.363,170.630,34.398,156.467
C01202=1048.919,72.251,418.345,170.631,34.399,156.467
C01203=1048.925,72.500,418.327,170.633,34.401,156.467
C01204=1048.931,72.749,418.309,170.635,34.403,156.467
C01205=1048.937,72.999,418.291,170.636,34.405,156.468
C01206=1048.944,73.248,418.273,170.638,34.407,156.468
C01207=1048.949,73.497,418.255,170.640,34.409,156.468
C01208=1048.955,73.746,418.236,170.641,34.411,156.469
C01209=1048.962,73.996,418.219,170.644,34.413,156.469
C01210=1048.968,74.245,418.200,170.645,34.414,156.469
C01211=1048.974,74.494,418.182,170.647,34.416,156.470
C01212=1048.980,74.743,418.164,170.649,34.418,156.470
C01213=1048.987,74.993,418.146,170.650,34.420,156.470
C01214=1048.993,75.242,418.128,170.652,34.422,156.471
C01215=1048.999,75.492,418.110,170.654,34.424,156.471
C01216=1049.005,75.740,418.091,170.655,34.425,156.471
C01217=1049.011,75.990,418.074,170.657,34.427,156.472
C01218=1049.018,76.239,418.055,170.658,34.429,156.472
C01219=1049.024,76.488,418.036,170.660,34.431,156.472
C01220=1049.030,76.738,418.018,170.662,34.433,156.472
C01221=1049.036,76.986,418.000,170.663,34.435,156.473
C01222=1049.044,77.272,417.979,170.665,34.437,156.473
C01223=1049.050,77.558,417.958,170.668,34.439,156.474
C01224=1049.057,77.844,417.938,170.670,34.441,156.474
C01225=1049.065,78.130,417.916,170.672,34.443,156.474
C01226=1049.071,78.379,417.897,170.673,34.445,156.475
C01227=1049.077,78.628,417.880,170.675,34.447,156.475
C01228=1049.083,78.877,417.861,170.677,34.449,156.475
C01229=1049.089,79.126,417.843,170.678,34.451,156.476
C01230=1049.095,79.377,417.824,170.680,34.453,156.476
C01231=1049.101,79.626,417.805,170.681,34.455,156.476
C01232=1049.108,79.875,417.787,170.683,34.457,156.477
C01233=1049.113,80.123,417.768,170.685,34.459,156.477
C01234=1049.120,80.373,417.751,170.686,34.460,156.477
C01235=1049.125,80.622,417.731,170.689,34.462,156.478
C01236=1049.132,80.872,417.713,170.690,34.464,156.478
C01237=1049.138,81.121,417.695,170.692,34.466,156.478
C01238=1049.144,81.370,417.676,170.694,34.468,156.479
C01239=1049.150,81.619,417.658,170.695,34.470,156.479
C01240=1049.156,81.868,417.639,170.697,34.472,156.479
C01241=1049.162,82.118,417.621,170.699,34.473,156.479
C01242=1049.168,82.367,417.602,170.700,34.475,156.480
C01243=1049.175,82.616,417.583,170.702,34.477,156.480
C01244=1049.181,82.865,417.565,170.703,34.479,156.480
C01245=1049.187,83.115,417.545,170.705,34.481,156.481
C01246=1049.192,83.364,417.528,170.707,34.483,156.481
C01247=1049.199,83.613,417.509,170.708,34.485,156.481
C01248=1049.205,83.862,417.491,170.711,34.487,156.482
C01249=1049.212,84.111,417.472,170.712,34.489,156.482
C01250=1049.217,84.361,417.453,170.714,34.491,156.482
C01251=1049.223,84.610,417.435,170.716,34.493,156.483
C01252=1049.230,84.859,417.416,170.717,34.495,156.483
C01253=1049.236,85.109,417.397,170.719,34.497,156.483
C01254=1049.242,85.358,417.378,170.721,34.499,156.484
C01255=1049.248,85.607,417.360,170.722,34.500,156.484
C01256=1049.255,85.856,417.341,170.724,34.502,156.484
C01257=1049.261,86.105,417.322,170.725,34.504,156.485
C01258=1049.267,86.354,417.305,170.727,34.506,156.485
C01259=1049.272,86.604,417.285,170.729,34.508,156.485
C01260=1049.279,86.853,417.267,170.731,34.509,156.486
C01261=1049.285,87.102,417.248,170.733,34.511,156.486
C01262=1049.292,87.351,417.230,170.735,34.513,156.486
C01263=1049.297,87.601,417.210,170.736,34.515,156.487
C01264=1049.304,87.850,417.192,170.738,34.517,156.487
C01265=1049.310,88.099,417.173,170.740,34.519,156.487
C01266=1049.317,88.348,417.154,170.741,34.521,156.488
C01267=1049.322,88.597,417.135,170.743,34.523,156.488
C01268=1049.329,88.847,417.116,170.744,34.524,156.488
C01269=1049.335,89.096,417.098,170.746,34.526,156.488
C01270=1049.342,89.345,417.079,170.748,34.528,156.489
C01271=1049.347,89.594,417.060,170.749,34.530,156.489
C01272=1049.354,89.843,417.041,170.752,34.532,156.489
C01273=1049.360,90.092,417.023,170.754,34.534,156.490
C01274=1049.366,90.342,417.003,170.755,34.536,156.490
C01275=1049.372,90.591,416.985,170.757,34.538,156.490
C01276=1049.379,90.840,416.966,170.759,34.540,156.491
C01277=1049.384,91.090,416.947,170.760,34.542,156.491
C01278=1049.391,91.339,416.928,170.762,34.544,156.491
C01279=1049.397,91.588,416.909,170.763,34.546,156.492
C01280=1049.402,91.838,416.890,170.765,34.547,156.492
C01281=1049.409,92.087,416.871,170.767,34.549,156.492
C01282=1049.414,92.336,416.852,170.768,34.551,156.493
C01283=1049.421,92.585,416.832,170.770,34.553,156.493
C01284=1049.427,92.834,416.813,170.772,34.555,156.493
C01285=1049.433,93.083,416.795,170.774,34.557,156.494
C01286=1049.440,93.370,416.773,170.776,34.559,156.494
C01287=1049.447,93.655,416.751,170.778,34.562,156.494
C01288=1049.454,93.941,416.729,170.780,34.564,156.495
C01289=1049.461,94.226,416.707,170.782,34.566,156.495
C01290=1049.467,94.475,416.688,170.783,34.568,156.496
C01291=1049.473,94.724,416.669,170.785,34.570,156.496
C01292=1049.479,94.974,416.650,170.786,34.572,156.496
C01293=1049.486,95.222,416.631,170.788,34.574,156.497
C01294=1049.492,95.472,416.611,170.791,34.576,156.497
C01295=1049.498,95.722,416.592,170.792,34.578,156.497
C01296=1049.504,95.971,416.573,170.794,34.580,156.498
C01297=1049.510,96.220,416.553,170.796,34.582,156.498
C01298=1049.517,96.469,416.535,170.797,34.583,156.498
C01299=1049.522,96.718,416.515,170.799,34.585,156.499
C01300=1049.529,96.968,416.497,170.801,34.587,156.499
C01301=1049.535,97.216,416.477,170.802,34.589,156.499
C01302=1049.541,97.465,416.458,170.804,34.591,156.500
C01303=1049.547,97.715,416.439,170.806,34.593,156.500
C01304=1049.553,97.964,416.420,170.807,34.595,156.500
C01305=1049.559,98.213,416.400,170.810,34.597,156.501
C01306=1049.565,98.462,416.381,170.811,34.599,156.501
C01307=1049.572,98.712,416.362,170.813,34.601,156.501
C01308=1049.578,98.961,416.342,170.815,34.603,156.502
C01309=1049.584,99.210,416.323,170.816,34.605,156.502
C01310=1049.590,99.459,416.304,170.818,34.607,156.502
C01311=1049.597,99.708,416.285,170.820,34.608,156.502
C01312=1049.602,99.957,416.266,170.821,34.610,156.503
C01313=1049.608,100.207,416.246,170.823,34.612,156.503
C01314=1049.615,100.456,416.227,170.825,34.614,156.503
C01315=1049.621,100.705,416.207,170.826,34.616,156.504
C01316=1049.628,100.955,416.189,170.828,34.617,156.504
C01317=1049.634,101.203,416.169,170.831,34.620,156.505
C01318=1049.639,101.453,416.150,170.832,34.622,156.505
C01319=1049.645,101.702,416.130,170.834,34.624,156.505
C01320=1049.651,101.951,416.110,170.835,34.626,156.506
C01321=1049.657,102.200,416.090,170.837,34.628,156.506
C01322=1049.663,102.449,416.072,170.839,34.630,156.506
C01323=1049.670,102.699,416.051,170.840,34.632,156.507
C01324=1049.676,102.948,416.032,170.842,34.633,156.507
C01325=1049.682,103.197,416.012,170.844,34.635,156.507
C01326=1049.687,103.446,415.993,170.845,34.637,156.508
C01327=1049.694,103.695,415.974,170.848,34.639,156.508
C01328=1049.700,103.944,415.954,170.850,34.641,156.508
C01329=1049.706,104.193,415.934,170.851,34.643,156.509
C01330=1049.712,104.443,415.915,170.853,34.646,156.509
C01331=1049.718,104.692,415.895,170.855,34.648,156.509
C01332=1049.724,104.941,415.876,170.856,34.649,156.510
C01333=1049.730,105.190,415.856,170.858,34.651,156.510
C01334=1049.736,105.439,415.837,170.860,34.653,156.510
C01335=1049.742,105.688,415.817,170.861,34.655,156.511
C01336=1049.749,105.938,415.797,170.863,34.657,156.511
C01337=1049.754,106.187,415.777,170.865,34.659,156.511
C01338=1049.761,106.435,415.758,170.867,34.661,156.512
C01339=1049.767,106.685,415.739,170.869,34.663,156.512
C01340=1049.773,106.934,415.719,170.870,34.665,156.512
C01341=1049.779,107.183,415.699,170.872,34.667,156.513
C01342=1049.785,107.433,415.679,170.874,34.669,156.513
C01343=1049.791,107.682,415.659,170.875,34.671,156.513
C01344=1049.797,107.931,415.640,170.877,34.673,156.514
C01345=1049.803,108.179,415.621,170.879,34.674,156.514
C01346=1049.810,108.429,415.600,170.880,34.676,156.514
C01347=1049.816,108.678,415.581,170.882,34.678,156.515
C01348=1049.822,108.927,415.561,170.885,34.680,156.515
C01349=1049.828,109.176,415.541,170.886,34.683,156.516
C01350=1049.835,109.462,415.519,170.888,34.685,156.516
C01351=1049.842,109.748,415.496,170.890,34.687,156.516
C01352=1049.849,110.033,415.474,170.892,34.689,156.517
C01353=1049.856,110.319,415.451,170.894,34.691,156.517
C01354=1049.862,110.555,415.432,170.896,34.693,156.517
C01355=1049.867,110.790,415.414,170.897,34.695,156.518
C01356=1049.874,111.025,415.395,170.899,34.697,156.518
C01357=1049.880,111.260,415.376,170.901,34.699,156.518
C01358=1049.886,111.495,415.357,170.903,34.701,156.519
C01359=1049.891,111.730,415.339,170.905,34.703,156.519
C01360=1049.897,111.965,415.319,170.906,34.704,156.519
C01361=1049.902,112.201,415.301,170.908,34.706,156.520
C01362=1049.908,112.450,415.281,170.909,34.708,156.520
C01363=1049.914,112.699,415.261,170.911,34.710,156.520
C01364=1049.920,112.947,415.241,170.913,34.712,156.521
C01365=1049.927,113.197,415.220,170.914,34.714,156.521
C01366=1049.933,113.446,415.201,170.916,34.716,156.521
C01367=1049.939,113.695,415.181,170.918,34.718,156.522
C01368=1049.945,113.945,415.161,170.921,34.720,156.522
C01369=1049.951,114.193,415.141,170.922,34.722,156.522
C01370=1049.957,114.443,415.120,170.924,34.724,156.523
C01371=1049.963,114.691,415.100,170.925,34.726,156.523
C01372=1049.969,114.941,415.080,170.927,34.728,156.523
C01373=1049.975,115.190,415.060,170.929,34.730,156.524
C01374=1049.980,115.439,415.040,170.930,34.732,156.524
C01375=1049.986,115.688,415.020,170.932,34.734,156.525
C01376=1049.993,115.937,414.999,170.934,34.736,156.525
C01377=1049.999,116.186,414.979,170.936,34.738,156.525
C01378=1050.004,116.436,414.960,170.938,34.740,156.526
C01379=1050.011,116.685,414.939,170.940,34.743,156.526
C01380=1050.017,116.934,414.919,170.941,34.745,156.526
C01381=1050.022,117.183,414.899,170.943,34.747,156.527
C01382=1050.028,117.432,414.879,170.945,34.748,156.527
C01383=1050.035,117.681,414.858,170.947,34.750,156.527
C01384=1050.041,117.930,414.838,170.948,34.753,156.528
C01385=1050.046,118.179,414.817,170.950,34.755,156.528
C01386=1050.052,118.428,414.797,170.953,34.757,156.529
C01387=1050.058,118.677,414.777,170.954,34.759,156.529
C01388=1050.064,118.926,414.757,170.956,34.761,156.529
C01389=1050.070,119.176,414.736,170.958,34.763,156.530
C01390=1050.076,119.425,414.716,170.959,34.765,156.530
C01391=1050.082,119.673,414.696,170.961,34.767,156.530
C01392=1050.088,119.923,414.675,170.963,34.769,156.531
C01393=1050.094,120.172,414.655,170.964,34.771,156.531
C01394=1050.101,120.422,414.635,170.966,34.773,156.531
C01395=1050.106,120.671,414.614,170.969,34.775,156.532
C01396=1050.112,120.920,414.594,170.970,34.777,156.532
C01397=1050.119,121.168,414.573,170.972,34.779,156.532
C01398=1050.125,121.417,414.553,170.974,34.781,156.533
C01399=1050.130,121.666,414.533,170.976,34.783,156.533
C01400=1050.137,121.916,414.513,170.977,34.785,156.533
C01401=1050.143,122.165,414.493,170.979,34.787,156.534
C01402=1050.149,122.415,414.472,170.981,34.789,156.534
C01403=1050.155,122.663,414.451,170.982,34.791,156.535
C01404=1050.161,122.912,414.431,170.984,34.793,156.535
C01405=1050.167,123.161,414.410,170.987,34.795,156.535
C01406=1050.173,123.410,414.390,170.989,34.797,156.536
C01407=1050.179,123.660,414.370,170.990,34.799,156.536
C01408=1050.185,123.908,414.349,170.992,34.801,156.536
C01409=1050.192,124.158,414.328,170.994,34.803,156.537
C01410=1050.198,124.407,414.308,170.995,34.805,156.537
C01411=1050.203,124.656,414.288,170.997,34.807,156.537
C01412=1050.210,124.905,414.267,170.999,34.809,156.538
C01413=1050.216,125.153,414.247,171.002,34.811,156.538
C01414=1050.224,125.468,414.220,171.004,34.814,156.539
C01415=1050.231,125.781,414.195,171.006,34.816,156.539
C01416=1050.239,126.094,414.169,171.008,34.818,156.539
C01417=1050.247,126.409,414.143,171.010,34.821,156.540
C01418=1050.253,126.657,414.122,171.012,34.823,156.540
C01419=1050.258,126.906,414.102,171.014,34.825,156.541
C01420=1050.265,127.155,414.082,171.015,34.827,156.541
C01421=1050.271,127.405,414.061,171.018,34.829,156.541
C01422=1050.277,127.653,414.040,171.020,34.831,156.542
C01423=1050.284,127.903,414.020,171.022,34.833,156.542
C01424=1050.289,128.151,413.998,171.023,34.835,156.542
C01425=1050.296,128.401,413.978,171.025,34.837,156.543
C01426=1050.302,128.650,413.958,171.027,34.839,156.543
C01427=1050.308,128.899,413.936,171.029,34.841,156.544
C01428=1050.314,129.148,413.917,171.030,34.843,156.544
C01429=1050.321,129.397,413.896,171.032,34.845,156.544
C01430=1050.326,129.646,413.875,171.035,34.847,156.545
C01431=1050.333,129.895,413.855,171.037,34.849,156.545
C01432=1050.338,130.144,413.833,171.038,34.851,156.545
C01433=1050.345,130.393,413.813,171.040,34.853,156.546
C01434=1050.352,130.642,413.792,171.042,34.855,156.546
C01435=1050.357,130.891,413.771,171.044,34.857,156.546
C01436=1050.364,131.141,413.751,171.045,34.859,156.547
C01437=1050.370,131.389,413.730,171.047,34.861,156.547
C01438=1050.376,131.639,413.709,171.049,34.863,156.547
C01439=1050.381,131.887,413.688,171.052,34.865,156.548
C01440=1050.388,132.137,413.668,171.053,34.867,156.548
C01441=1050.394,132.386,413.646,171.055,34.869,156.548
C01442=1050.400,132.635,413.625,171.057,34.871,156.549
C01443=1050.406,132.884,413.605,171.059,34.874,156.549
C01444=1050.412,133.133,413.583,171.060,34.876,156.550
C01445=1050.418,133.382,413.562,171.062,34.877,156.550
C01446=1050.424,133.631,413.542,171.064,34.879,156.550
C01447=1050.430,133.880,413.521,171.067,34.882,156.551
C01448=1050.435,134.129,413.500,171.068,34.884,156.551
C01449=1050.442,134.378,413.479,171.070,34.886,156.551
C01450=1050.448,134.628,413.458,171.072,34.888,156.552
C01451=1050.454,134.876,413.436,171.074,34.890,156.552
C01452=1050.461,135.125,413.415,171.075,34.892,156.553
C01453=1050.466,135.374,413.395,171.077,34.894,156.553
C01454=1050.472,135.623,413.373,171.079,34.896,156.553
C01455=1050.479,135.872,413.352,171.081,34.898,156.554
C01456=1050.484,136.121,413.332,171.084,34.900,156.554
C01457=1050.490,136.371,413.310,171.085,34.902,156.554
C01458=1050.496,136.619,413.289,171.087,34.904,156.555
C01459=1050.502,136.869,413.268,171.089,34.907,156.555
C01460=1050.509,137.118,413.247,171.091,34.908,156.556
C01461=1050.514,137.366,413.225,171.092,34.910,156.556
C01462=1050.521,137.616,413.205,171.094,34.912,156.556
C01463=1050.527,137.865,413.183,171.096,34.915,156.557
C01464=1050.533,138.114,413.162,171.099,34.917,156.557
C01465=1050.539,138.363,413.141,171.101,34.919,156.557
C01466=1050.545,138.612,413.121,171.102,34.921,156.558
C01467=1050.551,138.861,413.099,171.104,34.923,156.558
C01468=1050.557,139.110,413.077,171.106,34.925,156.558
C01469=1050.563,139.359,413.056,171.108,34.927,156.559
C01470=1050.569,139.608,413.034,171.109,34.929,156.559
C01471=1050.575,139.857,413.014,171.111,34.931,156.560
C01472=1050.581,140.106,412.993,171.114,34.933,156.560
C01473=1050.587,140.355,412.971,171.116,34.936,156.560
C01474=1050.593,140.604,412.950,171.118,34.938,156.561
C01475=1050.599,140.853,412.928,171.119,34.939,156.561
C01476=1050.605,141.102,412.907,171.121,34.942,156.562
C01477=1050.611,141.351,412.885,171.123,34.944,156.562
C01478=1050.618,141.636,412.861,171.125,34.946,156.562
C01479=1050.625,141.922,412.836,171.128,34.949,156.563
C01480=1050.631,142.207,412.812,171.130,34.951,156.563
C01481=1050.639,142.493,412.787,171.132,34.953,156.564
C01482=1050.644,142.741,412.766,171.134,34.956,156.564
C01483=1050.651,142.990,412.745,171.136,34.958,156.564
C01484=1050.657,143.240,412.723,171.138,34.960,156.565
C01485=1050.662,143.488,412.702,171.139,34.962,156.565
C01486=1050.668,143.737,412.680,171.141,34.964,156.566
C01487=1050.675,143.987,412.658,171.144,34.966,156.566
C01488=1050.681,144.236,412.637,171.146,34.968,156.566
C01489=1050.686,144.484,412.615,171.148,34.970,156.567
C01490=1050.693,144.734,412.594,171.149,34.972,156.567
C01491=1050.699,144.983,412.572,171.151,34.975,156.567
C01492=1050.704,145.231,412.551,171.153,34.977,156.568
C01493=1050.710,145.480,412.529,171.155,34.979,156.568
C01494=1050.717,145.730,412.508,171.158,34.981,156.569
C01495=1050.723,145.979,412.486,171.160,34.983,156.569
C01496=1050.729,146.228,412.464,171.161,34.985,156.569
C01497=1050.735,146.476,412.444,171.163,34.987,156.570
C01498=1050.741,146.725,412.422,171.165,34.989,156.570
C01499=1050.748,146.975,412.400,171.167,34.991,156.570
C01500=1050.754,147.224,412.379,171.169,34.994,156.571
C01501=1050.759,147.472,412.358,171.171,34.996,156.571
C01502=1050.765,147.722,412.336,171.173,34.998,156.572
C01503=1050.771,147.970,412.313,171.175,35.000,156.572
C01504=1050.777,148.220,412.291,171.177,35.002,156.572
C01505=1050.783,148.468,412.270,171.179,35.004,156.573
C01506=1050.789,148.717,412.248,171.181,35.006,156.573
C01507=1050.795,148.967,412.227,171.183,35.009,156.574
C01508=1050.801,149.216,412.205,171.184,35.011,156.574
C01509=1050.808,149.464,412.183,171.186,35.013,156.574
C01510=1050.813,149.713,412.161,171.189,35.015,156.575
C01511=1050.819,149.962,412.139,171.191,35.017,156.575
C01512=1050.825,150.212,412.118,171.193,35.020,156.576
C01513=1050.831,150.460,412.095,171.195,35.021,156.576
C01514=1050.838,150.709,412.074,171.196,35.024,156.576
C01515=1050.843,150.958,412.052,171.198,35.026,156.577
C01516=1050.849,151.207,412.030,171.200,35.028,156.577
C01517=1050.855,151.456,412.008,171.203,35.030,156.578
C01518=1050.861,151.705,411.986,171.205,35.032,156.578
C01519=1050.867,151.954,411.965,171.207,35.035,156.578
C01520=1050.874,152.204,411.943,171.208,35.036,156.579
C01521=1050.879,152.452,411.920,171.210,35.039,156.579
C01522=1050.885,152.701,411.899,171.212,35.041,156.579
C01523=1050.891,152.950,411.877,171.214,35.043,156.580
C01524=1050.897,153.199,411.855,171.217,35.045,156.580
C01525=1050.904,153.448,411.833,171.219,35.047,156.581
C01526=1050.909,153.697,411.810,171.221,35.050,156.581
C01527=1050.915,153.945,411.789,171.223,35.052,156.581
C01528=1050.921,154.195,411.767,171.224,35.054,156.582
C01529=1050.928,154.443,411.745,171.226,35.056,156.582
C01530=1050.933,154.693,411.723,171.228,35.058,156.583
C01531=1050.939,154.942,411.701,171.231,35.060,156.583
C01532=1050.946,155.191,411.679,171.233,35.063,156.583
C01533=1050.951,155.440,411.656,171.235,35.065,156.584
C01534=1050.958,155.689,411.634,171.237,35.067,156.584
C01535=1050.964,155.938,411.612,171.239,35.069,156.585
C01536=1050.969,156.186,411.590,171.240,35.072,156.585
C01537=1050.975,156.435,411.568,171.242,35.074,156.585
C01538=1050.981,156.684,411.546,171.245,35.076,156.586
C01539=1050.987,156.933,411.524,171.247,35.078,156.586
C01540=1050.993,157.182,411.501,171.249,35.080,156.587
C01541=1050.999,157.431,411.480,171.251,35.082,156.587
C01542=1051.006,157.716,411.453,171.253,35.085,156.588
C01543=1051.013,158.002,411.428,171.255,35.087,156.588
C01544=1051.019,158.287,411.403,171.258,35.090,156.588
C01545=1051.026,158.571,411.377,171.261,35.092,156.589
C01546=1051.032,158.820,411.356,171.262,35.095,156.589
C01547=1051.038,159.069,411.333,171.264,35.097,156.590
C01548=1051.045,159.318,411.310,171.266,35.099,156.590
C01549=1051.051,159.567,411.289,171.268,35.101,156.591
C01550=1051.057,159.816,411.266,171.270,35.104,156.591
C01551=1051.063,160.065,411.244,171.273,35.106,156.591
C01552=1051.069,160.314,411.222,171.275,35.108,156.592
C01553=1051.075,160.563,411.199,171.277,35.110,156.592
C01554=1051.081,160.812,411.177,171.279,35.112,156.593
C01555=1051.087,161.061,411.154,171.281,35.114,156.593
C01556=1051.093,161.310,411.131,171.282,35.117,156.593
C01557=1051.098,161.559,411.109,171.285,35.119,156.594
C01558=1051.104,161.808,411.087,171.287,35.121,156.594
C01559=1051.110,162.057,411.064,171.289,35.124,156.595
C01560=1051.116,162.306,411.041,171.291,35.126,156.595
C01561=1051.121,162.555,411.019,171.293,35.129,156.596
C01562=1051.128,162.804,410.996,171.295,35.131,156.596
C01563=1051.133,163.052,410.974,171.297,35.133,156.596
C01564=1051.139,163.301,410.951,171.300,35.136,156.597
C01565=1051.144,163.550,410.928,171.302,35.138,156.597
C01566=1051.150,163.799,410.906,171.303,35.140,156.598
C01567=1051.156,164.048,410.883,171.305,35.142,156.598
C01568=1051.162,164.297,410.860,171.307,35.144,156.598
C01569=1051.168,164.546,410.837,171.309,35.147,156.599
C01570=1051.173,164.794,410.814,171.312,35.149,156.599
C01571=1051.180,165.043,410.792,171.314,35.152,156.600
C01572=1051.186,165.292,410.769,171.316,35.154,156.600
C01573=1051.191,165.541,410.747,171.318,35.156,156.601
C01574=1051.197,165.790,410.724,171.320,35.159,156.601
C01575=1051.203,166.039,410.701,171.322,35.161,156.601
C01576=1051.209,166.288,410.679,171.325,35.163,156.602
C01577=1051.215,166.537,410.656,171.327,35.166,156.602
C01578=1051.220,166.786,410.633,171.329,35.168,156.603
C01579=1051.226,167.035,410.610,171.330,35.170,156.603
C01580=1051.232,167.283,410.587,171.332,35.172,156.604
C01581=1051.238,167.532,410.565,171.334,35.175,156.604
C01582=1051.244,167.781,410.542,171.337,35.177,156.604
C01583=1051.250,168.030,410.519,171.339,35.179,156.605
C01584=1051.256,168.279,410.496,171.341,35.182,156.605
C01585=1051.261,168.528,410.473,171.343,35.184,156.606
C01586=1051.268,168.776,410.450,171.345,35.186,156.606
C01587=1051.274,169.026,410.427,171.347,35.189,156.607
C01588=1051.280,169.275,410.404,171.350,35.191,156.607
C01589=1051.286,169.524,410.381,171.352,35.193,156.608
C01590=1051.291,169.772,410.358,171.354,35.196,156.608
C01591=1051.298,170.021,410.336,171.356,35.198,156.608
C01592=1051.304,170.270,410.313,171.358,35.200,156.609
C01593=1051.309,170.519,410.290,171.360,35.202,156.609
C01594=1051.315,170.768,410.267,171.362,35.205,156.610
C01595=1051.321,171.017,410.244,171.365,35.207,156.610
C01596=1051.326,171.266,410.221,171.367,35.209,156.611
C01597=1051.333,171.515,410.198,171.369,35.212,156.611
C01598=1051.340,171.763,410.175,171.371,35.214,156.611
C01599=1051.345,172.012,410.152,171.373,35.216,156.612
C01600=1051.351,172.261,410.129,171.375,35.219,156.612
C01601=1051.357,172.510,410.106,171.378,35.221,156.613
C01602=1051.362,172.759,410.083,171.380,35.224,156.613
C01603=1051.369,173.008,410.060,171.382,35.226,156.614
C01604=1051.376,173.256,410.037,171.384,35.228,156.614
C01605=1051.381,173.505,410.014,171.386,35.230,156.614
C01606=1051.387,173.790,409.987,171.389,35.233,156.615
C01607=1051.395,174.075,409.961,171.391,35.235,156.615
C01608=1051.401,174.359,409.934,171.394,35.239,156.616
C01609=1051.408,174.644,409.909,171.396,35.241,156.616
C01610=1051.415,174.893,409.885,171.398,35.244,156.617
C01611=1051.421,175.142,409.862,171.400,35.245,156.617
C01612=1051.426,175.390,409.839,171.403,35.248,156.618
C01613=1051.432,175.639,409.816,171.405,35.250,156.618
C01614=1051.439,175.888,409.792,171.407,35.252,156.619
C01615=1051.444,176.137,409.769,171.409,35.255,156.619
C01616=1051.451,176.386,409.747,171.411,35.257,156.619
C01617=1051.457,176.635,409.724,171.413,35.260,156.620
C01618=1051.463,176.884,409.700,171.416,35.262,156.620
C01619=1051.469,177.133,409.677,171.418,35.264,156.621
C01620=1051.475,177.381,409.654,171.420,35.267,156.621
C01621=1051.481,177.630,409.630,171.422,35.269,156.622
C01622=1051.487,177.879,409.607,171.425,35.271,156.622
C01623=1051.493,178.128,409.583,171.427,35.273,156.622
C01624=1051.499,178.377,409.560,171.430,35.276,156.623
C01625=1051.506,178.626,409.537,171.432,35.278,156.623
C01626=1051.512,178.874,409.514,171.434,35.280,156.624
C01627=1051.518,179.123,409.491,171.436,35.283,156.624
C01628=1051.524,179.372,409.467,171.438,35.285,156.625
C01629=1051.530,179.621,409.444,171.441,35.288,156.625
C01630=1051.536,179.870,409.421,171.443,35.290,156.626
C01631=1051.542,180.119,409.397,171.445,35.292,156.626
C01632=1051.548,180.368,409.374,171.447,35.295,156.626
C01633=1051.554,180.616,409.350,171.449,35.297,156.627
C01634=1051.561,180.866,409.327,171.451,35.299,156.627
C01635=1051.567,181.114,409.303,171.454,35.301,156.628
C01636=1051.572,181.363,409.280,171.457,35.304,156.628
C01637=1051.580,181.611,409.257,171.459,35.306,156.629
C01638=1051.585,181.860,409.234,171.461,35.308,156.629
C01639=1051.591,182.109,409.210,171.463,35.311,156.629
C01640=1051.598,182.358,409.187,171.465,35.313,156.630
C01641=1051.604,182.606,409.163,171.468,35.316,156.630
C01642=1051.610,182.856,409.140,171.470,35.318,156.631
C01643=1051.616,183.104,409.116,171.472,35.320,156.631
C01644=1051.622,183.353,409.093,171.474,35.323,156.632
C01645=1051.629,183.602,409.069,171.476,35.325,156.632
C01646=1051.635,183.850,409.046,171.480,35.327,156.633
C01647=1051.641,184.100,409.022,171.482,35.329,156.633
C01648=1051.647,184.348,408.999,171.484,35.332,156.633
C01649=1051.652,184.597,408.974,171.486,35.334,156.634
C01650=1051.659,184.846,408.951,171.488,35.337,156.634
C01651=1051.664,185.095,408.927,171.490,35.339,156.635
C01652=1051.670,185.343,408.903,171.493,35.342,156.635
C01653=1051.676,185.593,408.879,171.495,35.345,156.636
C01654=1051.682,185.842,408.856,171.497,35.347,156.636
C01655=1051.688,186.090,408.832,171.499,35.350,156.637
C01656=1051.694,186.339,408.807,171.501,35.352,156.637
C01657=1051.700,186.587,408.784,171.504,35.355,156.638
C01658=1051.705,186.836,408.759,171.507,35.357,156.638
C01659=1051.711,187.086,408.736,171.509,35.360,156.639
C01660=1051.716,187.334,408.712,171.511,35.362,156.639
C01661=1051.723,187.583,408.688,171.513,35.365,156.640
C01662=1051.728,187.832,408.664,171.516,35.367,156.640
C01663=1051.734,188.080,408.640,171.518,35.370,156.641
C01664=1051.740,188.329,408.615,171.520,35.372,156.641
C01665=1051.746,188.578,408.592,171.522,35.375,156.642
C01666=1051.752,188.826,408.567,171.524,35.378,156.642
C01667=1051.758,189.076,408.544,171.528,35.380,156.643
C01668=1051.763,189.324,408.520,171.530,35.383,156.643
C01669=1051.770,189.573,408.496,171.532,35.385,156.644
C01670=1051.777,189.857,408.468,171.534,35.388,156.644
C01671=1051.784,190.142,408.441,171.537,35.391,156.645
C01672=1051.790,190.426,408.414,171.540,35.394,156.645
C01673=1051.797,190.710,408.385,171.543,35.397,156.646
C01674=1051.803,190.959,408.361,171.545,35.399,156.646
C01675=1051.808,191.207,408.337,171.547,35.402,156.647
C01676=1051.815,191.456,408.313,171.550,35.404,156.647
C01677=1051.820,191.705,408.289,171.552,35.407,156.648
C01678=1051.827,191.954,408.265,171.554,35.409,156.648
C01679=1051.832,192.202,408.241,171.556,35.412,156.649
C01680=1051.839,192.451,408.217,171.559,35.414,156.649
C01681=1051.844,192.700,408.192,171.562,35.417,156.650
C01682=1051.851,192.949,408.168,171.564,35.420,156.650
C01683=1051.856,193.197,408.144,171.566,35.422,156.651
C01684=1051.863,193.446,408.120,171.568,35.425,156.651
C01685=1051.868,193.695,408.096,171.570,35.427,156.652
C01686=1051.875,193.943,408.071,171.574,35.430,156.652
C01687=1051.881,194.193,408.046,171.576,35.432,156.653
C01688=1051.887,194.441,408.023,171.578,35.434,156.653
C01689=1051.893,194.690,407.998,171.580,35.437,156.653
C01690=1051.899,194.939,407.974,171.582,35.440,156.654
C01691=1051.905,195.188,407.950,171.586,35.443,156.655
C01692=1051.911,195.436,407.926,171.588,35.445,156.655
C01693=1051.917,195.685,407.901,171.590,35.447,156.655
C01694=1051.923,195.934,407.876,171.592,35.450,156.656
C01695=1051.929,196.182,407.853,171.594,35.452,156.656
C01696=1051.935,196.432,407.828,171.598,35.455,156.657
C01697=1051.941,196.679,407.804,171.600,35.458,156.657
C01698=1051.947,196.929,407.779,171.602,35.460,156.658
C01699=1051.954,197.178,407.755,171.604,35.463,156.658
C01700=1051.959,197.426,407.731,171.607,35.465,156.659
C01701=1051.966,197.674,407.706,171.610,35.468,156.659
C01702=1051.971,197.923,407.682,171.612,35.471,156.660
C01703=1051.977,198.172,407.657,171.614,35.473,156.660
C01704=1051.984,198.421,407.633,171.616,35.476,156.661
C01705=1051.989,198.669,407.608,171.620,35.478,156.661
C01706=1051.996,198.918,407.584,171.622,35.481,156.662
C01707=1052.002,199.168,407.559,171.624,35.483,156.662
C01708=1052.007,199.416,407.534,171.626,35.486,156.663
C01709=1052.014,199.665,407.510,171.629,35.489,156.663
C01710=1052.020,199.914,407.486,171.632,35.491,156.664
C01711=1052.027,200.162,407.461,171.634,35.494,156.664
C01712=1052.032,200.411,407.437,171.636,35.496,156.665
C01713=1052.039,200.659,407.412,171.639,35.499,156.665
C01714=1052.045,200.908,407.387,171.642,35.502,156.666
C01715=1052.050,201.157,407.363,171.644,35.504,156.666
C01716=1052.057,201.405,407.338,171.646,35.507,156.667
C01717=1052.063,201.655,407.314,171.649,35.509,156.667
C01718=1052.069,201.903,407.288,171.651,35.512,156.668
C01719=1052.075,202.152,407.264,171.654,35.515,156.668
C01720=1052.081,202.401,407.239,171.656,35.518,156.669
C01721=1052.088,202.650,407.215,171.659,35.520,156.669
C01722=1052.093,202.898,407.190,171.661,35.523,156.670
C01723=1052.099,203.146,407.164,171.664,35.526,156.670
C01724=1052.105,203.395,407.140,171.666,35.528,156.671
C01725=1052.111,203.643,407.115,171.669,35.531,156.672
C01726=1052.117,203.893,407.090,171.671,35.534,156.672
C01727=1052.123,204.141,407.065,171.673,35.536,156.673
C01728=1052.129,204.390,407.040,171.676,35.539,156.673
C01729=1052.134,204.639,407.015,171.679,35.542,156.674
C01730=1052.141,204.887,406.990,171.681,35.545,156.674
C01731=1052.147,205.136,406.965,171.683,35.547,156.675
C01732=1052.153,205.384,406.941,171.687,35.550,156.675
C01733=1052.159,205.633,406.916,171.689,35.553,156.676
C01734=1052.184,206.686,406.810,171.909,35.647,156.693
C01735=1052.191,206.932,406.784,171.911,35.651,156.694
C01736=1052.198,207.178,406.758,171.912,35.654,156.694
C01737=1052.204,207.426,406.732,171.915,35.657,156.695
C01738=1052.210,207.671,406.707,171.917,35.661,156.696
C01739=1052.216,207.919,406.681,171.918,35.665,156.696
C01740=1052.222,208.165,406.655,171.921,35.668,156.697
C01741=1052.229,208.412,406.629,171.923,35.672,156.698
C01742=1052.235,208.659,406.603,171.924,35.675,156.698
C01743=1052.242,208.907,406.577,171.926,35.678,156.699
C01744=1052.247,209.155,406.551,171.929,35.682,156.700
C01745=1052.254,209.405,406.525,171.930,35.686,156.701
C01746=1052.261,209.653,406.499,171.933,35.689,156.701
C01747=1052.267,209.901,406.473,171.934,35.693,156.702
C01748=1052.273,210.151,406.446,171.936,35.696,156.703
C01749=1052.280,210.399,406.420,171.938,35.699,156.703
C01750=1052.286,210.647,406.394,171.940,35.703,156.704
C01751=1052.293,210.896,406.367,171.942,35.707,156.705
C01752=1052.299,211.144,406.342,171.945,35.710,156.706
C01753=1052.305,211.393,406.315,171.946,35.714,156.706
C01754=1052.312,211.642,406.289,171.948,35.717,156.707
C01755=1052.318,211.890,406.263,171.950,35.721,156.708
C01756=1052.324,212.139,406.237,171.953,35.724,156.708
C01757=1052.331,212.387,406.211,171.954,35.728,156.709
C01758=1052.337,212.636,406.184,171.957,35.731,156.710
C01759=1052.343,212.884,406.158,171.959,35.735,156.711
C01760=1052.350,213.133,406.131,171.960,35.739,156.711
C01761=1052.356,213.381,406.105,171.963,35.742,156.712
C01762=1052.362,213.629,406.078,171.965,35.745,156.713
C01763=1052.369,213.879,406.052,171.966,35.749,156.713
C01764=1052.375,214.127,406.026,171.969,35.752,156.714
C01765=1052.381,214.375,406.000,171.971,35.756,156.715
C01766=1052.387,214.624,405.973,171.972,35.760,156.716
C01767=1052.393,214.872,405.946,171.975,35.763,156.716
C01768=1052.400,215.121,405.920,171.977,35.766,156.717
C01769=1052.406,215.370,405.893,171.979,35.770,156.718
C01770=1052.413,215.618,405.867,171.981,35.773,156.718
C01771=1052.419,215.867,405.840,171.983,35.777,156.719
C01772=1052.425,216.115,405.814,171.985,35.781,156.720
C01773=1052.432,216.364,405.787,171.987,35.784,156.720
C01774=1052.438,216.612,405.761,171.989,35.787,156.721
C01775=1052.444,216.860,405.734,171.991,35.791,156.722
C01776=1052.450,217.109,405.707,171.994,35.794,156.723
C01777=1052.457,217.357,405.681,171.995,35.798,156.723
C01778=1052.463,217.606,405.654,171.997,35.801,156.724
C01779=1052.470,217.854,405.628,172.000,35.805,156.725
C01780=1052.476,218.103,405.601,172.002,35.808,156.725
C01781=1052.483,218.351,405.575,172.003,35.812,156.726
C01782=1052.489,218.601,405.548,172.006,35.815,156.727
C01783=1052.495,218.849,405.521,172.008,35.818,156.728
C01784=1052.502,219.097,405.494,172.010,35.822,156.728
C01785=1052.508,219.345,405.468,172.012,35.826,156.729
C01786=1052.515,219.594,405.441,172.014,35.829,156.730
C01787=1052.521,219.843,405.414,172.016,35.832,156.730
C01788=1052.527,220.092,405.387,172.019,35.836,156.731
C01789=1052.534,220.340,405.361,172.020,35.839,156.732
C01790=1052.540,220.589,405.334,172.022,35.842,156.732
C01791=1052.547,220.838,405.307,172.025,35.846,156.733
C01792=1052.553,221.088,405.280,172.027,35.850,156.734
C01793=1052.559,221.339,405.253,172.030,35.853,156.735
C01794=1052.565,221.589,405.225,172.031,35.857,156.735
C01795=1052.572,221.837,405.199,172.033,35.860,156.736
C01796=1052.578,222.086,405.172,172.036,35.863,156.737
C01797=1052.584,222.334,405.146,172.038,35.867,156.737
C01798=1052.591,222.583,405.118,172.039,35.871,156.738
C01799=1052.597,222.831,405.091,172.042,35.874,156.739
C01800=1052.603,223.080,405.064,172.044,35.877,156.740
C01801=1052.610,223.328,405.037,172.046,35.881,156.740
C01802=1052.616,223.577,405.011,172.049,35.884,156.741
C01803=1052.623,223.826,404.984,172.050,35.888,156.742
C01804=1052.629,224.074,404.956,172.052,35.891,156.742
C01805=1052.635,224.323,404.929,172.055,35.895,156.743
C01806=1052.641,224.571,404.903,172.057,35.898,156.744
C01807=1052.648,224.819,404.875,172.059,35.902,156.745
C01808=1052.654,225.068,404.849,172.061,35.905,156.745
C01809=1052.661,225.316,404.821,172.063,35.908,156.746
C01810=1052.667,225.565,404.794,172.066,35.912,156.747
C01811=1052.673,225.813,404.767,172.068,35.916,156.747
C01812=1052.679,226.062,404.740,172.070,35.919,156.748
C01813=1052.685,226.310,404.713,172.073,35.922,156.749
